LIN {X 0,Y 390.032,Z 462.401,A -85,B 0,C 180,E1 -11489.872,E2 -11489.872} C_VEL
LIN {X 0,Y 390.019,Z 462.384,A -85,B 0,C 180,E1 -11493.227,E2 -11493.227} C_VEL
LIN {X 0,Y 390.057,Z 462.395,A -85,B 0,C 180,E1 -11496.766,E2 -11496.766} C_VEL
LIN {X 0,Y 390.061,Z 462.376,A -85,B 0,C 180,E1 -11499.983,E2 -11499.983} C_VEL
LIN {X 0,Y 390.074,Z 462.387,A -85,B 0,C 180,E1 -11503.247,E2 -11503.247} C_VEL
LIN {X 0,Y 390.188,Z 462.376,A -85,B 0,C 180,E1 -11506.563,E2 -11506.563} C_VEL
LIN {X 0,Y 390.178,Z 462.363,A -85,B 0,C 180,E1 -11510.672,E2 -11510.672} C_VEL
LIN {X 0,Y 390.269,Z 462.37,A -85,B 0,C 180,E1 -11513.799,E2 -11513.799} C_VEL
LIN {X 0,Y 390.398,Z 462.338,A -85,B 0,C 180,E1 -11517.938,E2 -11517.938} C_VEL
LIN {X 0,Y 390.398,Z 462.347,A -85,B 0,C 180,E1 -11522.065,E2 -11522.065} C_VEL
LIN {X 0,Y 390.271,Z 462.365,A -85,B 0,C 180,E1 -11526.204,E2 -11526.204} C_VEL
LIN {X 0,Y 390.181,Z 462.355,A -85,B 0,C 180,E1 -11529.331,E2 -11529.331} C_VEL
LIN {X 0,Y 390.151,Z 462.381,A -85,B 0,C 180,E1 -11532.485,E2 -11532.485} C_VEL
LIN {X 0,Y 390.051,Z 462.394,A -85,B 0,C 180,E1 -11535.682,E2 -11535.682} C_VEL
LIN {X 0,Y 390.037,Z 462.377,A -85,B 0,C 180,E1 -11538.927,E2 -11538.927} C_VEL
LIN {X 0,Y 390.029,Z 462.4,A -85,B 0,C 180,E1 -11542.236,E2 -11542.236} C_VEL
LIN {X 0,Y 390.05,Z 462.383,A -85,B 0,C 180,E1 -11545.723,E2 -11545.723} C_VEL
LIN {X 0,Y 390.023,Z 462.396,A -85,B 0,C 180,E1 -11549.114,E2 -11549.114} C_VEL
LIN {X 0,Y 390.041,Z 462.389,A -85,B 0,C 180,E1 -11552.723,E2 -11552.723} C_VEL
LIN {X 0,Y 390.042,Z 462.395,A -85,B 0,C 180,E1 -11555.823,E2 -11555.823} C_VEL
LIN {X 0,Y 390.034,Z 462.394,A -85,B 0,C 180,E1 -11559.213,E2 -11559.213} C_VEL
LIN {X 0,Y 390.03,Z 462.4,A -85,B 0,C 180,E1 -11562.373,E2 -11562.373} C_VEL
LIN {X 0,Y 390.039,Z 462.397,A -85,B 0,C 180,E1 -11565.354,E2 -11565.354} C_VEL
LIN {X 0,Y 390.013,Z 462.387,A -85,B 0,C 180,E1 -11568.185,E2 -11568.185} C_VEL
LIN {X 0,Y 390.056,Z 462.395,A -85,B 0,C 180,E1 -11570.904,E2 -11570.904} C_VEL
LIN {X 0,Y 390.07,Z 462.391,A -85,B 0,C 180,E1 -11574.792,E2 -11574.792} C_VEL
LIN {X 0,Y 390.024,Z 462.406,A -85,B 0,C 180,E1 -11578.496,E2 -11578.496} C_VEL
LIN {X 0,Y 390.119,Z 462.589,A -85,B 0,C 180,E1 -11579.67,E2 -11579.67} C_VEL
LIN {X 0,Y 392.065,Z 472.624,A -85,B 0,C 180,E1 -11582.8,E2 -11582.8} C_VEL
LIN {X 0,Y 392.806,Z 477.057,A -85,B 0,C 180,E1 -11584.071,E2 -11584.071} C_VEL
LIN {X 0,Y 392.549,Z 483.032,A -85,B 0,C 180,E1 -11585.684,E2 -11585.684} C_VEL
LIN {X 0,Y 391.661,Z 493.141,A -85,B 0,C 180,E1 -11588.417,E2 -11588.417} C_VEL
LIN {X 0,Y 391.382,Z 497.053,A -85,B 0,C 180,E1 -11589.469,E2 -11589.469} C_VEL
LIN {X 0,Y 391.927,Z 500.233,A -85,B 0,C 180,E1 -11589.618,E2 -11589.618} C_VEL
LIN {X 0,Y 396.826,Z 527.349,A -85,B 0,C 180,E1 -11590.388,E2 -11590.388} C_VEL
LIN {X 0,Y 395.882,Z 602.023,A -85,B 0,C 180,E1 -11591.767,E2 -11591.767} C_VEL
LIN {X 0,Y 395.479,Z 611.939,A -85,B 0,C 180,E1 -11592.049,E2 -11592.049} C_VEL
LIN {X 0,Y 395.02,Z 621.929,A -85,B 0,C 180,E1 -11592.462,E2 -11592.462} C_VEL
LIN {X 0,Y 394.399,Z 630.315,A -85,B 0,C 180,E1 -11592.901,E2 -11592.901} C_VEL
LIN {X 0,Y 393.654,Z 641.432,A -85,B 0,C 180,E1 -11593.669,E2 -11593.669} C_VEL
LIN {X 0,Y 392.916,Z 650.435,A -85,B 0,C 180,E1 -11594.437,E2 -11594.437} C_VEL
LIN {X 0,Y 392.266,Z 658.483,A -85,B 0,C 180,E1 -11595.259,E2 -11595.259} C_VEL
LIN {X 0,Y 391.546,Z 666.812,A -85,B 0,C 180,E1 -11596.274,E2 -11596.274} C_VEL
LIN {X 0,Y 390.769,Z 675.386,A -85,B 0,C 180,E1 -11597.536,E2 -11597.536} C_VEL
LIN {X 0,Y 390.167,Z 681.375,A -85,B 0,C 180,E1 -11598.572,E2 -11598.572} C_VEL
LIN {X 0,Y 389.667,Z 687.688,A -85,B 0,C 180,E1 -11599.872,E2 -11599.872} C_VEL
LIN {X 0,Y 389.264,Z 692.963,A -85,B 0,C 180,E1 -11601.172,E2 -11601.172} C_VEL
LIN {X 0,Y 388.944,Z 698.057,A -85,B 0,C 180,E1 -11602.734,E2 -11602.734} C_VEL
LIN {X 0,Y 388.73,Z 701.925,A -85,B 0,C 180,E1 -11604.248,E2 -11604.248} C_VEL
LIN {X 0,Y 388.702,Z 704.954,A -85,B 0,C 180,E1 -11605.853,E2 -11605.853} C_VEL
LIN {X 0,Y 388.636,Z 706.452,A -85,B 0,C 180,E1 -11606.89,E2 -11606.89} C_VEL
LIN {X 0,Y 388.705,Z 707.976,A -85,B 0,C 180,E1 -11608.964,E2 -11608.964} C_VEL
LIN {X 0,Y 388.709,Z 708.254,A -85,B 0,C 180,E1 -11610,E2 -11610} C_VEL
LIN {X 0,Y 388.663,Z 707.38,A -85,B 0,C 180,E1 -11612.073,E2 -11612.073} C_VEL
LIN {X 0,Y 388.636,Z 706.452,A -85,B 0,C 180,E1 -11613.11,E2 -11613.11} C_VEL
LIN {X 0,Y 388.744,Z 703.109,A -85,B 0,C 180,E1 -11615.186,E2 -11615.186} C_VEL
LIN {X 0,Y 388.848,Z 699.484,A -85,B 0,C 180,E1 -11616.747,E2 -11616.747} C_VEL
LIN {X 0,Y 389.146,Z 694.753,A -85,B 0,C 180,E1 -11618.307,E2 -11618.307} C_VEL
LIN {X 0,Y 389.578,Z 688.781,A -85,B 0,C 180,E1 -11619.868,E2 -11619.868} C_VEL
LIN {X 0,Y 390.051,Z 682.688,A -85,B 0,C 180,E1 -11621.168,E2 -11621.168} C_VEL
LIN {X 0,Y 390.631,Z 676.947,A -85,B 0,C 180,E1 -11622.204,E2 -11622.204} C_VEL
LIN {X 0,Y 391.252,Z 670.29,A -85,B 0,C 180,E1 -11623.24,E2 -11623.24} C_VEL
LIN {X 0,Y 391.877,Z 663.503,A -85,B 0,C 180,E1 -11624.15,E2 -11624.15} C_VEL
LIN {X 0,Y 392.529,Z 654.768,A -85,B 0,C 180,E1 -11625.14,E2 -11625.14} C_VEL
LIN {X 0,Y 393.366,Z 644.611,A -85,B 0,C 180,E1 -11626.077,E2 -11626.077} C_VEL
LIN {X 0,Y 394.089,Z 636.223,A -85,B 0,C 180,E1 -11626.712,E2 -11626.712} C_VEL
LIN {X 0,Y 394.727,Z 625.715,A -85,B 0,C 180,E1 -11627.351,E2 -11627.351} C_VEL
LIN {X 0,Y 395.28,Z 615.382,A -85,B 0,C 180,E1 -11627.827,E2 -11627.827} C_VEL
LIN {X 0,Y 395.748,Z 604.664,A -85,B 0,C 180,E1 -11628.173,E2 -11628.173} C_VEL
LIN {X 0,Y 396.177,Z 585.472,A -85,B 0,C 180,E1 -11628.554,E2 -11628.554} C_VEL
LIN {X 0,Y 396.727,Z 526.888,A -85,B 0,C 180,E1 -11629.626,E2 -11629.626} C_VEL
LIN {X 0,Y 391.632,Z 498.91,A -85,B 0,C 180,E1 -11630.424,E2 -11630.424} C_VEL
LIN {X 0,Y 391.346,Z 497.047,A -85,B 0,C 180,E1 -11630.533,E2 -11630.533} C_VEL
LIN {X 0,Y 392.557,Z 483.234,A -85,B 0,C 180,E1 -11634.316,E2 -11634.316} C_VEL
LIN {X 0,Y 392.862,Z 477.28,A -85,B 0,C 180,E1 -11635.937,E2 -11635.937} C_VEL
LIN {X 0,Y 391.203,Z 468.061,A -85,B 0,C 180,E1 -11638.625,E2 -11638.625} C_VEL
LIN {X 0,Y 390.098,Z 462.508,A -85,B 0,C 180,E1 -11640.369,E2 -11640.369} C_VEL
LIN {X 0,Y 390.072,Z 462.397,A -85,B 0,C 180,E1 -11644.024,E2 -11644.024} C_VEL
LIN {X 0,Y 390.036,Z 462.399,A -85,B 0,C 180,E1 -11647.78,E2 -11647.78} C_VEL
LIN {X 0,Y 390.016,Z 462.382,A -85,B 0,C 180,E1 -11650.813,E2 -11650.813} C_VEL
LIN {X 0,Y 390.042,Z 462.401,A -85,B 0,C 180,E1 -11653.883,E2 -11653.883} C_VEL
LIN {X 0,Y 390.048,Z 462.396,A -85,B 0,C 180,E1 -11656.787,E2 -11656.787} C_VEL
LIN {X 0,Y 390.01,Z 462.399,A -85,B 0,C 180,E1 -11659.553,E2 -11659.553} C_VEL
LIN {X 0,Y 390.037,Z 462.401,A -85,B 0,C 180,E1 -11662.45,E2 -11662.45} C_VEL
LIN {X 0,Y 390.062,Z 462.383,A -85,B 0,C 180,E1 -11666.043,E2 -11666.043} C_VEL
LIN {X 0,Y 390.043,Z 462.401,A -85,B 0,C 180,E1 -11669.869,E2 -11669.869} C_VEL
LIN {X 0,Y 390.029,Z 462.38,A -85,B 0,C 180,E1 -11673.224,E2 -11673.224} C_VEL
LIN {X 0,Y 390.058,Z 462.394,A -85,B 0,C 180,E1 -11676.766,E2 -11676.766} C_VEL
LIN {X 0,Y 390.066,Z 462.382,A -85,B 0,C 180,E1 -11679.98,E2 -11679.98} C_VEL
LIN {X 0,Y 390.076,Z 462.38,A -85,B 0,C 180,E1 -11683.244,E2 -11683.244} C_VEL
LIN {X 0,Y 390.13,Z 462.384,A -85,B 0,C 180,E1 -11686.599,E2 -11686.599} C_VEL
LIN {X 0,Y 390.152,Z 462.367,A -85,B 0,C 180,E1 -11689.621,E2 -11689.621} C_VEL
LIN {X 0,Y 390.242,Z 462.365,A -85,B 0,C 180,E1 -11692.756,E2 -11692.756} C_VEL
LIN {X 0,Y 390.193,Z 462.378,A -85,B 0,C 180,E1 -11694.832,E2 -11694.832} C_VEL
LIN {X 0,Y 390.399,Z 462.347,A -85,B 0,C 180,E1 -11697.935,E2 -11697.935} C_VEL
LIN {X 0,Y 390.398,Z 462.338,A -85,B 0,C 180,E1 -11702.062,E2 -11702.062} C_VEL
LIN {X 0,Y 390.247,Z 462.37,A -85,B 0,C 180,E1 -11706.515,E2 -11706.515} C_VEL
LIN {X 0,Y 390.178,Z 462.363,A -85,B 0,C 180,E1 -11709.328,E2 -11709.328} C_VEL
LIN {X 0,Y 390.188,Z 462.376,A -85,B 0,C 180,E1 -11713.437,E2 -11713.437} C_VEL
LIN {X 0,Y 390.063,Z 462.388,A -85,B 0,C 180,E1 -11717.269,E2 -11717.269} C_VEL
LIN {X 0,Y 390.041,Z 462.389,A -85,B 0,C 180,E1 -11721.121,E2 -11721.121} C_VEL
LIN {X 0,Y 390.033,Z 462.397,A -85,B 0,C 180,E1 -11724.482,E2 -11724.482} C_VEL
LIN {X 0,Y 390.005,Z 462.387,A -85,B 0,C 180,E1 -11727.996,E2 -11727.996} C_VEL
LIN {X 0,Y 390.01,Z 462.403,A -85,B 0,C 180,E1 -11731.503,E2 -11731.503} C_VEL
LIN {X 0,Y 390.056,Z 462.384,A -85,B 0,C 180,E1 -11735.207,E2 -11735.207} C_VEL
LIN {X 0,Y 390.044,Z 462.395,A -85,B 0,C 180,E1 -11739.095,E2 -11739.095} C_VEL
LIN {X 0,Y 390.017,Z 462.403,A -85,B 0,C 180,E1 -11742.371,E2 -11742.371} C_VEL
LIN {X 0,Y 390.026,Z 462.395,A -85,B 0,C 180,E1 -11745.352,E2 -11745.352} C_VEL
LIN {X 0,Y 389.997,Z 462.37,A -85,B 0,C 180,E1 -11748.183,E2 -11748.183} C_VEL
LIN {X 0,Y 390.039,Z 462.397,A -85,B 0,C 180,E1 -11750.902,E2 -11750.902} C_VEL
LIN {X 0,Y 390.053,Z 462.376,A -85,B 0,C 180,E1 -11754.79,E2 -11754.79} C_VEL
LIN {X 0,Y 390.006,Z 462.404,A -85,B 0,C 180,E1 -11758.495,E2 -11758.495} C_VEL
LIN {X 0,Y 390,Z 462.399,A -85,B 0,C 180,E1 -11762.002,E2 -11762.002} C_VEL
LIN {X 0,Y 390.027,Z 462.403,A -85,B 0,C 180,E1 -11765.516,E2 -11765.516} C_VEL
LIN {X 0,Y 390.04,Z 462.401,A -85,B 0,C 180,E1 -11768.877,E2 -11768.877} C_VEL
LIN {X 0,Y 390.087,Z 462.397,A -85,B 0,C 180,E1 -11772.165,E2 -11772.165} C_VEL
LIN {X 0,Y 390.076,Z 462.398,A -85,B 0,C 180,E1 -11775.39,E2 -11775.39} C_VEL
LIN {X 0,Y 390.151,Z 462.389,A -85,B 0,C 180,E1 -11777.516,E2 -11777.516} C_VEL
LIN {X 0,Y 390.197,Z 462.441,A -85,B 0,C 180,E1 -11781.324,E2 -11781.324} C_VEL
LIN {X 0,Y 390.388,Z 463.13,A -85,B 0,C 180,E1 -11782.098,E2 -11782.098} C_VEL
LIN {X 0,Y 391.792,Z 466.011,A -85,B 0,C 180,E1 -11783.369,E2 -11783.369} C_VEL
LIN {X 0,Y 393.843,Z 467.786,A -85,B 0,C 180,E1 -11785.138,E2 -11785.138} C_VEL
LIN {X 0,Y 395.352,Z 468.399,A -85,B 0,C 180,E1 -11786.943,E2 -11786.943} C_VEL
LIN {X 0,Y 396.116,Z 469.029,A -85,B 0,C 180,E1 -11788.983,E2 -11788.983} C_VEL
LIN {X 0,Y 396.296,Z 469.069,A -85,B 0,C 180,E1 -11790,E2 -11790} C_VEL
LIN {X 0,Y 395.957,Z 468.754,A -85,B 0,C 180,E1 -11791.78,E2 -11791.78} C_VEL
LIN {X 0,Y 394.887,Z 468.274,A -85,B 0,C 180,E1 -11793.622,E2 -11793.622} C_VEL
LIN {X 0,Y 393.539,Z 467.583,A -85,B 0,C 180,E1 -11795.123,E2 -11795.123} C_VEL
LIN {X 0,Y 391.792,Z 466.011,A -85,B 0,C 180,E1 -11796.631,E2 -11796.631} C_VEL
LIN {X 0,Y 390.503,Z 463.555,A -85,B 0,C 180,E1 -11797.722,E2 -11797.722} C_VEL
LIN {X 0,Y 390.256,Z 462.638,A -85,B 0,C 180,E1 -11798.283,E2 -11798.283} C_VEL
LIN {X 0,Y 390.121,Z 462.392,A -85,B 0,C 180,E1 -11801.429,E2 -11801.429} C_VEL
LIN {X 0,Y 390.153,Z 462.388,A -85,B 0,C 180,E1 -11803.543,E2 -11803.543} C_VEL
LIN {X 0,Y 390.092,Z 462.395,A -85,B 0,C 180,E1 -11807.288,E2 -11807.288} C_VEL
LIN {X 0,Y 390.072,Z 462.398,A -85,B 0,C 180,E1 -11810.47,E2 -11810.47} C_VEL
LIN {X 0,Y 390.047,Z 462.401,A -85,B 0,C 180,E1 -11813.353,E2 -11813.353} C_VEL
LIN {X 0,Y 390.015,Z 462.403,A -85,B 0,C 180,E1 -11816.775,E2 -11816.775} C_VEL
LIN {X 0,Y 390.021,Z 462.393,A -85,B 0,C 180,E1 -11820.301,E2 -11820.301} C_VEL
LIN {X 0,Y 389.994,Z 462.397,A -85,B 0,C 180,E1 -11820.778,E2 -11820.778} C_VEL
LIN {X 0,Y 389.32,Z 462.491,A -85,B 0,C 180,E1 -11821.641,E2 -11821.641} C_VEL
LIN {X 0,Y 386.473,Z 462.838,A -85,B 0,C 180,E1 -11823.042,E2 -11823.042} C_VEL
LIN {X 0,Y 384.074,Z 463.124,A -85,B 0,C 180,E1 -11824.175,E2 -11824.175} C_VEL
LIN {X 0,Y 383.052,Z 463.246,A -85,B 0,C 180,E1 -11825.051,E2 -11825.051} C_VEL
LIN {X 0,Y 382.973,Z 463.257,A -85,B 0,C 180,E1 -11825.348,E2 -11825.348} C_VEL
LIN {X 0,Y 382.963,Z 463.279,A -85,B 0,C 180,E1 -11828.605,E2 -11828.605} C_VEL
LIN {X 0,Y 382.945,Z 463.25,A -85,B 0,C 180,E1 -11831.352,E2 -11831.352} C_VEL
LIN {X 0,Y 382.974,Z 463.266,A -85,B 0,C 180,E1 -11834.303,E2 -11834.303} C_VEL
LIN {X 0,Y 382.969,Z 463.279,A -85,B 0,C 180,E1 -11837.237,E2 -11837.237} C_VEL
LIN {X 0,Y 382.972,Z 463.277,A -85,B 0,C 180,E1 -11840.421,E2 -11840.421} C_VEL
LIN {X 0,Y 383.001,Z 463.268,A -85,B 0,C 180,E1 -11844.044,E2 -11844.044} C_VEL
LIN {X 0,Y 382.974,Z 463.276,A -85,B 0,C 180,E1 -11847.58,E2 -11847.58} C_VEL
LIN {X 0,Y 382.964,Z 463.275,A -85,B 0,C 180,E1 -11850.3,E2 -11850.3} C_VEL
LIN {X 0,Y 382.993,Z 463.267,A -85,B 0,C 180,E1 -11854.047,E2 -11854.047} C_VEL
LIN {X 0,Y 382.979,Z 463.278,A -85,B 0,C 180,E1 -11857.335,E2 -11857.335} C_VEL
LIN {X 0,Y 383.003,Z 463.251,A -85,B 0,C 180,E1 -11860.715,E2 -11860.715} C_VEL
LIN {X 0,Y 383.002,Z 463.276,A -85,B 0,C 180,E1 -11864.025,E2 -11864.025} C_VEL
LIN {X 0,Y 383.127,Z 463.255,A -85,B 0,C 180,E1 -11867.285,E2 -11867.285} C_VEL
LIN {X 0,Y 383.129,Z 463.238,A -85,B 0,C 180,E1 -11870.499,E2 -11870.499} C_VEL
LIN {X 0,Y 383.227,Z 463.246,A -85,B 0,C 180,E1 -11873.684,E2 -11873.684} C_VEL
LIN {X 0,Y 383.363,Z 463.214,A -85,B 0,C 180,E1 -11877.9,E2 -11877.9} C_VEL
LIN {X 0,Y 383.363,Z 463.223,A -85,B 0,C 180,E1 -11882.103,E2 -11882.103} C_VEL
LIN {X 0,Y 383.229,Z 463.241,A -85,B 0,C 180,E1 -11886.319,E2 -11886.319} C_VEL
LIN {X 0,Y 383.171,Z 463.23,A -85,B 0,C 180,E1 -11888.439,E2 -11888.439} C_VEL
LIN {X 0,Y 383.079,Z 463.254,A -85,B 0,C 180,E1 -11891.644,E2 -11891.644} C_VEL
LIN {X 0,Y 383.05,Z 463.27,A -85,B 0,C 180,E1 -11893.8,E2 -11893.8} C_VEL
LIN {X 0,Y 383.02,Z 463.256,A -85,B 0,C 180,E1 -11897.421,E2 -11897.421} C_VEL
LIN {X 0,Y 383.01,Z 463.267,A -85,B 0,C 180,E1 -11900.641,E2 -11900.641} C_VEL
LIN {X 0,Y 383.007,Z 463.274,A -85,B 0,C 180,E1 -11903.81,E2 -11903.81} C_VEL
LIN {X 0,Y 382.968,Z 463.26,A -85,B 0,C 180,E1 -11907.31,E2 -11907.31} C_VEL
LIN {X 0,Y 382.981,Z 463.276,A -85,B 0,C 180,E1 -11910.92,E2 -11910.92} C_VEL
LIN {X 0,Y 383.012,Z 463.265,A -85,B 0,C 180,E1 -11914.67,E2 -11914.67} C_VEL
LIN {X 0,Y 382.991,Z 463.277,A -85,B 0,C 180,E1 -11917.903,E2 -11917.903} C_VEL
LIN {X 0,Y 382.961,Z 463.278,A -85,B 0,C 180,E1 -11921.352,E2 -11921.352} C_VEL
LIN {X 0,Y 382.989,Z 463.273,A -85,B 0,C 180,E1 -11924.303,E2 -11924.303} C_VEL
LIN {X 0,Y 382.982,Z 463.277,A -85,B 0,C 180,E1 -11927.237,E2 -11927.237} C_VEL
LIN {X 0,Y 382.986,Z 463.269,A -85,B 0,C 180,E1 -11930.42,E2 -11930.42} C_VEL
LIN {X 0,Y 383.014,Z 463.264,A -85,B 0,C 180,E1 -11934.044,E2 -11934.044} C_VEL
LIN {X 0,Y 382.985,Z 463.272,A -85,B 0,C 180,E1 -11937.58,E2 -11937.58} C_VEL
LIN {X 0,Y 383.068,Z 463.508,A -85,B 0,C 180,E1 -11939.384,E2 -11939.384} C_VEL
LIN {X 0,Y 385.013,Z 473.48,A -85,B 0,C 180,E1 -11942.554,E2 -11942.554} C_VEL
LIN {X 0,Y 385.9,Z 479.744,A -85,B 0,C 180,E1 -11944.372,E2 -11944.372} C_VEL
LIN {X 0,Y 384.943,Z 490.991,A -85,B 0,C 180,E1 -11947.456,E2 -11947.456} C_VEL
LIN {X 0,Y 384.447,Z 496.846,A -85,B 0,C 180,E1 -11949.081,E2 -11949.081} C_VEL
LIN {X 0,Y 385.014,Z 500.013,A -85,B 0,C 180,E1 -11949.235,E2 -11949.235} C_VEL
LIN {X 0,Y 389.987,Z 527.524,A -85,B 0,C 180,E1 -11950.037,E2 -11950.037} C_VEL
LIN {X 0,Y 389.957,Z 544.905,A -85,B 0,C 180,E1 -11950.368,E2 -11950.368} C_VEL
LIN {X 0,Y 389.156,Z 601.827,A -85,B 0,C 180,E1 -11951.44,E2 -11951.44} C_VEL
LIN {X 0,Y 388.725,Z 611.743,A -85,B 0,C 180,E1 -11951.726,E2 -11951.726} C_VEL
LIN {X 0,Y 388.253,Z 621.733,A -85,B 0,C 180,E1 -11952.146,E2 -11952.146} C_VEL
LIN {X 0,Y 387.504,Z 632.088,A -85,B 0,C 180,E1 -11952.723,E2 -11952.723} C_VEL
LIN {X 0,Y 386.829,Z 641.235,A -85,B 0,C 180,E1 -11953.373,E2 -11953.373} C_VEL
LIN {X 0,Y 386.047,Z 650.238,A -85,B 0,C 180,E1 -11954.153,E2 -11954.153} C_VEL
LIN {X 0,Y 385.326,Z 658.968,A -85,B 0,C 180,E1 -11955.071,E2 -11955.071} C_VEL
LIN {X 0,Y 384.598,Z 666.804,A -85,B 0,C 180,E1 -11956.048,E2 -11956.048} C_VEL
LIN {X 0,Y 383.824,Z 675.189,A -85,B 0,C 180,E1 -11957.307,E2 -11957.307} C_VEL
LIN {X 0,Y 383.183,Z 681.178,A -85,B 0,C 180,E1 -11958.361,E2 -11958.361} C_VEL
LIN {X 0,Y 382.663,Z 687.492,A -85,B 0,C 180,E1 -11959.685,E2 -11959.685} C_VEL
LIN {X 0,Y 382.219,Z 692.766,A -85,B 0,C 180,E1 -11961.008,E2 -11961.008} C_VEL
LIN {X 0,Y 381.873,Z 697.86,A -85,B 0,C 180,E1 -11962.598,E2 -11962.598} C_VEL
LIN {X 0,Y 381.674,Z 701.247,A -85,B 0,C 180,E1 -11963.907,E2 -11963.907} C_VEL
LIN {X 0,Y 381.627,Z 704.758,A -85,B 0,C 180,E1 -11965.776,E2 -11965.776} C_VEL
LIN {X 0,Y 381.548,Z 706.256,A -85,B 0,C 180,E1 -11966.832,E2 -11966.832} C_VEL
LIN {X 0,Y 381.604,Z 707.779,A -85,B 0,C 180,E1 -11968.945,E2 -11968.945} C_VEL
LIN {X 0,Y 381.623,Z 708.059,A -85,B 0,C 180,E1 -11970,E2 -11970} C_VEL
LIN {X 0,Y 381.561,Z 707.183,A -85,B 0,C 180,E1 -11972.111,E2 -11972.111} C_VEL
LIN {X 0,Y 381.548,Z 706.256,A -85,B 0,C 180,E1 -11973.168,E2 -11973.168} C_VEL
LIN {X 0,Y 381.644,Z 702.912,A -85,B 0,C 180,E1 -11975.283,E2 -11975.283} C_VEL
LIN {X 0,Y 381.785,Z 699.287,A -85,B 0,C 180,E1 -11976.872,E2 -11976.872} C_VEL
LIN {X 0,Y 382.099,Z 694.556,A -85,B 0,C 180,E1 -11978.461,E2 -11978.461} C_VEL
LIN {X 0,Y 382.541,Z 688.584,A -85,B 0,C 180,E1 -11980.051,E2 -11980.051} C_VEL
LIN {X 0,Y 383.064,Z 682.491,A -85,B 0,C 180,E1 -11981.375,E2 -11981.375} C_VEL
LIN {X 0,Y 383.647,Z 676.75,A -85,B 0,C 180,E1 -11982.43,E2 -11982.43} C_VEL
LIN {X 0,Y 384.311,Z 670.093,A -85,B 0,C 180,E1 -11983.483,E2 -11983.483} C_VEL
LIN {X 0,Y 385.024,Z 662.625,A -85,B 0,C 180,E1 -11984.491,E2 -11984.491} C_VEL
LIN {X 0,Y 385.705,Z 654.177,A -85,B 0,C 180,E1 -11985.455,E2 -11985.455} C_VEL
LIN {X 0,Y 386.557,Z 644.415,A -85,B 0,C 180,E1 -11986.368,E2 -11986.368} C_VEL
LIN {X 0,Y 387.29,Z 636.027,A -85,B 0,C 180,E1 -11987.014,E2 -11987.014} C_VEL
LIN {X 0,Y 387.967,Z 625.519,A -85,B 0,C 180,E1 -11987.663,E2 -11987.663} C_VEL
LIN {X 0,Y 388.529,Z 615.186,A -85,B 0,C 180,E1 -11988.147,E2 -11988.147} C_VEL
LIN {X 0,Y 389.02,Z 604.468,A -85,B 0,C 180,E1 -11988.498,E2 -11988.498} C_VEL
LIN {X 0,Y 389.471,Z 583.485,A -85,B 0,C 180,E1 -11988.92,E2 -11988.92} C_VEL
LIN {X 0,Y 390.114,Z 528.302,A -85,B 0,C 180,E1 -11989.942,E2 -11989.942} C_VEL
LIN {X 0,Y 384.978,Z 500.003,A -85,B 0,C 180,E1 -11990.768,E2 -11990.768} C_VEL
LIN {X 0,Y 384.4,Z 497.123,A -85,B 0,C 180,E1 -11990.887,E2 -11990.887} C_VEL
LIN {X 0,Y 384.468,Z 495.674,A -85,B 0,C 180,E1 -11991.206,E2 -11991.206} C_VEL
LIN {X 0,Y 385.712,Z 483.045,A -85,B 0,C 180,E1 -11994.776,E2 -11994.776} C_VEL
LIN {X 0,Y 385.919,Z 478.968,A -85,B 0,C 180,E1 -11995.917,E2 -11995.917} C_VEL
LIN {X 0,Y 384.343,Z 469.806,A -85,B 0,C 180,E1 -11998.63,E2 -11998.63} C_VEL
LIN {X 0,Y 383.04,Z 463.38,A -85,B 0,C 180,E1 -12000.692,E2 -12000.692} C_VEL
LIN {X 0,Y 383.019,Z 463.277,A -85,B 0,C 180,E1 -12004.338,E2 -12004.338} C_VEL
LIN {X 0,Y 382.991,Z 463.274,A -85,B 0,C 180,E1 -12007.269,E2 -12007.269} C_VEL
LIN {X 0,Y 382.975,Z 463.264,A -85,B 0,C 180,E1 -12009.962,E2 -12009.962} C_VEL
LIN {X 0,Y 383.009,Z 463.273,A -85,B 0,C 180,E1 -12012.778,E2 -12012.778} C_VEL
LIN {X 0,Y 382.99,Z 463.273,A -85,B 0,C 180,E1 -12015.787,E2 -12015.787} C_VEL
LIN {X 0,Y 382.962,Z 463.277,A -85,B 0,C 180,E1 -12018.8,E2 -12018.8} C_VEL
LIN {X 0,Y 382.991,Z 463.277,A -85,B 0,C 180,E1 -12022.097,E2 -12022.097} C_VEL
LIN {X 0,Y 383.012,Z 463.265,A -85,B 0,C 180,E1 -12025.33,E2 -12025.33} C_VEL
LIN {X 0,Y 382.981,Z 463.276,A -85,B 0,C 180,E1 -12029.08,E2 -12029.08} C_VEL
LIN {X 0,Y 382.968,Z 463.26,A -85,B 0,C 180,E1 -12032.69,E2 -12032.69} C_VEL
LIN {X 0,Y 383.007,Z 463.274,A -85,B 0,C 180,E1 -12036.19,E2 -12036.19} C_VEL
LIN {X 0,Y 383.033,Z 463.265,A -85,B 0,C 180,E1 -12039.596,E2 -12039.596} C_VEL
LIN {X 0,Y 383.035,Z 463.257,A -85,B 0,C 180,E1 -12042.927,E2 -12042.927} C_VEL
LIN {X 0,Y 383.088,Z 463.262,A -85,B 0,C 180,E1 -12046.485,E2 -12046.485} C_VEL
LIN {X 0,Y 383.116,Z 463.245,A -85,B 0,C 180,E1 -12049.428,E2 -12049.428} C_VEL
LIN {X 0,Y 383.197,Z 463.242,A -85,B 0,C 180,E1 -12052.622,E2 -12052.622} C_VEL
LIN {X 0,Y 383.165,Z 463.254,A -85,B 0,C 180,E1 -12054.736,E2 -12054.736} C_VEL
LIN {X 0,Y 383.364,Z 463.223,A -85,B 0,C 180,E1 -12057.897,E2 -12057.897} C_VEL
LIN {X 0,Y 383.363,Z 463.214,A -85,B 0,C 180,E1 -12062.1,E2 -12062.1} C_VEL
LIN {X 0,Y 383.211,Z 463.246,A -85,B 0,C 180,E1 -12066.504,E2 -12066.504} C_VEL
LIN {X 0,Y 383.129,Z 463.238,A -85,B 0,C 180,E1 -12069.501,E2 -12069.501} C_VEL
LIN {X 0,Y 383.119,Z 463.257,A -85,B 0,C 180,E1 -12073.534,E2 -12073.534} C_VEL
LIN {X 0,Y 383.016,Z 463.267,A -85,B 0,C 180,E1 -12077.419,E2 -12077.419} C_VEL
LIN {X 0,Y 383.005,Z 463.264,A -85,B 0,C 180,E1 -12080.639,E2 -12080.639} C_VEL
LIN {X 0,Y 383.001,Z 463.278,A -85,B 0,C 180,E1 -12083.807,E2 -12083.807} C_VEL
LIN {X 0,Y 382.958,Z 463.262,A -85,B 0,C 180,E1 -12087.307,E2 -12087.307} C_VEL
LIN {X 0,Y 382.97,Z 463.279,A -85,B 0,C 180,E1 -12090.917,E2 -12090.917} C_VEL
LIN {X 0,Y 382.999,Z 463.262,A -85,B 0,C 180,E1 -12094.667,E2 -12094.667} C_VEL
LIN {X 0,Y 382.979,Z 463.282,A -85,B 0,C 180,E1 -12097.901,E2 -12097.901} C_VEL
LIN {X 0,Y 382.947,Z 463.271,A -85,B 0,C 180,E1 -12101.349,E2 -12101.349} C_VEL
LIN {X 0,Y 382.975,Z 463.277,A -85,B 0,C 180,E1 -12104.301,E2 -12104.301} C_VEL
LIN {X 0,Y 382.967,Z 463.248,A -85,B 0,C 180,E1 -12107.235,E2 -12107.235} C_VEL
LIN {X 0,Y 382.969,Z 463.271,A -85,B 0,C 180,E1 -12110.418,E2 -12110.418} C_VEL
LIN {X 0,Y 382.998,Z 463.261,A -85,B 0,C 180,E1 -12114.042,E2 -12114.042} C_VEL
LIN {X 0,Y 382.97,Z 463.278,A -85,B 0,C 180,E1 -12117.578,E2 -12117.578} C_VEL
LIN {X 0,Y 382.959,Z 463.266,A -85,B 0,C 180,E1 -12120.298,E2 -12120.298} C_VEL
LIN {X 0,Y 382.987,Z 463.281,A -85,B 0,C 180,E1 -12124.044,E2 -12124.044} C_VEL
LIN {X 0,Y 382.974,Z 463.282,A -85,B 0,C 180,E1 -12127.333,E2 -12127.333} C_VEL
LIN {X 0,Y 383.04,Z 463.274,A -85,B 0,C 180,E1 -12130.715,E2 -12130.715} C_VEL
LIN {X 0,Y 383.004,Z 463.279,A -85,B 0,C 180,E1 -12134.024,E2 -12134.024} C_VEL
LIN {X 0,Y 383.118,Z 463.264,A -85,B 0,C 180,E1 -12137.283,E2 -12137.283} C_VEL
LIN {X 0,Y 383.139,Z 463.583,A -85,B 0,C 180,E1 -12138.56,E2 -12138.56} C_VEL
LIN {X 0,Y 383.428,Z 464.757,A -85,B 0,C 180,E1 -12138.971,E2 -12138.971} C_VEL
LIN {X 0,Y 384.572,Z 466.794,A -85,B 0,C 180,E1 -12139.603,E2 -12139.603} C_VEL
LIN {X 0,Y 386.855,Z 468.647,A -85,B 0,C 180,E1 -12140.722,E2 -12140.722} C_VEL
LIN {X 0,Y 388.802,Z 469.821,A -85,B 0,C 180,E1 -12141.834,E2 -12141.834} C_VEL
LIN {X 0,Y 390.416,Z 472.61,A -85,B 0,C 180,E1 -12143.021,E2 -12143.021} C_VEL
LIN {X 0,Y 391.927,Z 474.117,A -85,B 0,C 180,E1 -12144.211,E2 -12144.211} C_VEL
LIN {X 0,Y 393.427,Z 475.106,A -85,B 0,C 180,E1 -12145.646,E2 -12145.646} C_VEL
LIN {X 0,Y 394.712,Z 475.569,A -85,B 0,C 180,E1 -12147.449,E2 -12147.449} C_VEL
LIN {X 0,Y 395.254,Z 476.076,A -85,B 0,C 180,E1 -12148.981,E2 -12148.981} C_VEL
LIN {X 0,Y 395.432,Z 476.106,A -85,B 0,C 180,E1 -12150,E2 -12150} C_VEL
LIN {X 0,Y 395.09,Z 475.808,A -85,B 0,C 180,E1 -12151.784,E2 -12151.784} C_VEL
LIN {X 0,Y 394.236,Z 475.37,A -85,B 0,C 180,E1 -12153.375,E2 -12153.375} C_VEL
LIN {X 0,Y 392.647,Z 474.648,A -85,B 0,C 180,E1 -12155.135,E2 -12155.135} C_VEL
LIN {X 0,Y 390.776,Z 473.066,A -85,B 0,C 180,E1 -12156.713,E2 -12156.713} C_VEL
LIN {X 0,Y 389.074,Z 470.321,A -85,B 0,C 180,E1 -12157.995,E2 -12157.995} C_VEL
LIN {X 0,Y 388.296,Z 469.392,A -85,B 0,C 180,E1 -12158.456,E2 -12158.456} C_VEL
LIN {X 0,Y 385.834,Z 468.03,A -85,B 0,C 180,E1 -12159.766,E2 -12159.766} C_VEL
LIN {X 0,Y 383.861,Z 465.743,A -85,B 0,C 180,E1 -12160.783,E2 -12160.783} C_VEL
LIN {X 0,Y 383.168,Z 463.833,A -85,B 0,C 180,E1 -12161.305,E2 -12161.305} C_VEL
LIN {X 0,Y 383.096,Z 463.3,A -85,B 0,C 180,E1 -12161.91,E2 -12161.91} C_VEL
LIN {X 0,Y 383.012,Z 463.278,A -85,B 0,C 180,E1 -12164.885,E2 -12164.885} C_VEL
LIN {X 0,Y 383.031,Z 463.275,A -85,B 0,C 180,E1 -12168.175,E2 -12168.175} C_VEL
LIN {X 0,Y 382.976,Z 463.282,A -85,B 0,C 180,E1 -12171.532,E2 -12171.532} C_VEL
LIN {X 0,Y 382.971,Z 463.281,A -85,B 0,C 180,E1 -12174.966,E2 -12174.966} C_VEL
LIN {X 0,Y 382.96,Z 463.269,A -85,B 0,C 180,E1 -12178.499,E2 -12178.499} C_VEL
LIN {X 0,Y 382.993,Z 463.277,A -85,B 0,C 180,E1 -12182.151,E2 -12182.151} C_VEL
LIN {X 0,Y 382.973,Z 463.257,A -85,B 0,C 180,E1 -12185.348,E2 -12185.348} C_VEL
LIN {X 0,Y 382.324,Z 463.351,A -85,B 0,C 180,E1 -12186.226,E2 -12186.226} C_VEL
LIN {X 0,Y 379.502,Z 463.713,A -85,B 0,C 180,E1 -12187.653,E2 -12187.653} C_VEL
LIN {X 0,Y 377.085,Z 464.012,A -85,B 0,C 180,E1 -12188.807,E2 -12188.807} C_VEL
LIN {X 0,Y 376.021,Z 464.135,A -85,B 0,C 180,E1 -12189.699,E2 -12189.699} C_VEL
LIN {X 0,Y 375.92,Z 464.141,A -85,B 0,C 180,E1 -12190.001,E2 -12190.001} C_VEL
LIN {X 0,Y 375.911,Z 464.136,A -85,B 0,C 180,E1 -12193.768,E2 -12193.768} C_VEL
LIN {X 0,Y 375.919,Z 464.157,A -85,B 0,C 180,E1 -12196.812,E2 -12196.812} C_VEL
LIN {X 0,Y 375.921,Z 464.156,A -85,B 0,C 180,E1 -12200.535,E2 -12200.535} C_VEL
LIN {X 0,Y 375.945,Z 464.155,A -85,B 0,C 180,E1 -12203.499,E2 -12203.499} C_VEL
LIN {X 0,Y 375.946,Z 464.142,A -85,B 0,C 180,E1 -12205.89,E2 -12205.89} C_VEL
LIN {X 0,Y 375.95,Z 464.157,A -85,B 0,C 180,E1 -12209.688,E2 -12209.688} C_VEL
LIN {X 0,Y 375.907,Z 464.141,A -85,B 0,C 180,E1 -12212.136,E2 -12212.136} C_VEL
LIN {X 0,Y 375.95,Z 464.154,A -85,B 0,C 180,E1 -12215.718,E2 -12215.718} C_VEL
LIN {X 0,Y 375.948,Z 464.144,A -85,B 0,C 180,E1 -12219.197,E2 -12219.197} C_VEL
LIN {X 0,Y 375.971,Z 464.144,A -85,B 0,C 180,E1 -12222.599,E2 -12222.599} C_VEL
LIN {X 0,Y 376.083,Z 464.134,A -85,B 0,C 180,E1 -12226.344,E2 -12226.344} C_VEL
LIN {X 0,Y 376.1,Z 464.111,A -85,B 0,C 180,E1 -12230.32,E2 -12230.32} C_VEL
LIN {X 0,Y 376.187,Z 464.122,A -85,B 0,C 180,E1 -12233.566,E2 -12233.566} C_VEL
LIN {X 0,Y 376.327,Z 464.09,A -85,B 0,C 180,E1 -12237.861,E2 -12237.861} C_VEL
LIN {X 0,Y 376.327,Z 464.1,A -85,B 0,C 180,E1 -12242.142,E2 -12242.142} C_VEL
LIN {X 0,Y 376.189,Z 464.116,A -85,B 0,C 180,E1 -12246.438,E2 -12246.438} C_VEL
LIN {X 0,Y 376.103,Z 464.107,A -85,B 0,C 180,E1 -12249.683,E2 -12249.683} C_VEL
LIN {X 0,Y 376.038,Z 464.141,A -85,B 0,C 180,E1 -12253.628,E2 -12253.628} C_VEL
LIN {X 0,Y 375.979,Z 464.13,A -85,B 0,C 180,E1 -12257.578,E2 -12257.578} C_VEL
LIN {X 0,Y 375.978,Z 464.143,A -85,B 0,C 180,E1 -12260.834,E2 -12260.834} C_VEL
LIN {X 0,Y 375.934,Z 464.149,A -85,B 0,C 180,E1 -12264.287,E2 -12264.287} C_VEL
LIN {X 0,Y 375.911,Z 464.137,A -85,B 0,C 180,E1 -12266.662,E2 -12266.662} C_VEL
LIN {X 0,Y 375.913,Z 464.154,A -85,B 0,C 180,E1 -12269.085,E2 -12269.085} C_VEL
LIN {X 0,Y 375.956,Z 464.155,A -85,B 0,C 180,E1 -12271.564,E2 -12271.564} C_VEL
LIN {X 0,Y 375.949,Z 464.146,A -85,B 0,C 180,E1 -12275.418,E2 -12275.418} C_VEL
LIN {X 0,Y 375.933,Z 464.152,A -85,B 0,C 180,E1 -12278.263,E2 -12278.263} C_VEL
LIN {X 0,Y 375.914,Z 464.158,A -85,B 0,C 180,E1 -12281.598,E2 -12281.598} C_VEL
LIN {X 0,Y 375.92,Z 464.155,A -85,B 0,C 180,E1 -12284.731,E2 -12284.731} C_VEL
LIN {X 0,Y 375.908,Z 464.15,A -85,B 0,C 180,E1 -12287.697,E2 -12287.697} C_VEL
LIN {X 0,Y 375.934,Z 464.149,A -85,B 0,C 180,E1 -12290.534,E2 -12290.534} C_VEL
LIN {X 0,Y 375.959,Z 464.143,A -85,B 0,C 180,E1 -12293.498,E2 -12293.498} C_VEL
LIN {X 0,Y 375.96,Z 464.155,A -85,B 0,C 180,E1 -12295.889,E2 -12295.889} C_VEL
LIN {X 0,Y 376.008,Z 464.333,A -85,B 0,C 180,E1 -12299.042,E2 -12299.042} C_VEL
LIN {X 0,Y 377.99,Z 474.336,A -85,B 0,C 180,E1 -12302.301,E2 -12302.301} C_VEL
LIN {X 0,Y 378.956,Z 480.604,A -85,B 0,C 180,E1 -12304.163,E2 -12304.163} C_VEL
LIN {X 0,Y 378.053,Z 490.795,A -85,B 0,C 180,E1 -12307.022,E2 -12307.022} C_VEL
LIN {X 0,Y 377.522,Z 496.692,A -85,B 0,C 180,E1 -12308.686,E2 -12308.686} C_VEL
LIN {X 0,Y 378.373,Z 501.077,A -85,B 0,C 180,E1 -12308.878,E2 -12308.878} C_VEL
LIN {X 0,Y 383.447,Z 529.25,A -85,B 0,C 180,E1 -12309.719,E2 -12309.719} C_VEL
LIN {X 0,Y 382.438,Z 601.631,A -85,B 0,C 180,E1 -12311.102,E2 -12311.102} C_VEL
LIN {X 0,Y 382.002,Z 611.547,A -85,B 0,C 180,E1 -12311.392,E2 -12311.392} C_VEL
LIN {X 0,Y 381.499,Z 621.536,A -85,B 0,C 180,E1 -12311.819,E2 -12311.819} C_VEL
LIN {X 0,Y 380.714,Z 631.891,A -85,B 0,C 180,E1 -12312.405,E2 -12312.405} C_VEL
LIN {X 0,Y 380.022,Z 641.039,A -85,B 0,C 180,E1 -12313.066,E2 -12313.066} C_VEL
LIN {X 0,Y 379.207,Z 650.041,A -85,B 0,C 180,E1 -12313.859,E2 -12313.859} C_VEL
LIN {X 0,Y 378.434,Z 658.771,A -85,B 0,C 180,E1 -12314.792,E2 -12314.792} C_VEL
LIN {X 0,Y 377.671,Z 666.788,A -85,B 0,C 180,E1 -12315.814,E2 -12315.814} C_VEL
LIN {X 0,Y 376.872,Z 674.992,A -85,B 0,C 180,E1 -12317.069,E2 -12317.069} C_VEL
LIN {X 0,Y 376.214,Z 680.982,A -85,B 0,C 180,E1 -12318.142,E2 -12318.142} C_VEL
LIN {X 0,Y 375.652,Z 687.295,A -85,B 0,C 180,E1 -12319.49,E2 -12319.49} C_VEL
LIN {X 0,Y 375.192,Z 692.569,A -85,B 0,C 180,E1 -12320.838,E2 -12320.838} C_VEL
LIN {X 0,Y 374.809,Z 697.663,A -85,B 0,C 180,E1 -12322.458,E2 -12322.458} C_VEL
LIN {X 0,Y 374.57,Z 701.388,A -85,B 0,C 180,E1 -12323.959,E2 -12323.959} C_VEL
LIN {X 0,Y 374.531,Z 704.562,A -85,B 0,C 180,E1 -12325.695,E2 -12325.695} C_VEL
LIN {X 0,Y 374.463,Z 706.06,A -85,B 0,C 180,E1 -12326.772,E2 -12326.772} C_VEL
LIN {X 0,Y 374.505,Z 707.583,A -85,B 0,C 180,E1 -12328.925,E2 -12328.925} C_VEL
LIN {X 0,Y 374.539,Z 707.863,A -85,B 0,C 180,E1 -12330,E2 -12330} C_VEL
LIN {X 0,Y 374.461,Z 706.987,A -85,B 0,C 180,E1 -12332.151,E2 -12332.151} C_VEL
LIN {X 0,Y 374.463,Z 706.06,A -85,B 0,C 180,E1 -12333.228,E2 -12333.228} C_VEL
LIN {X 0,Y 374.553,Z 702.716,A -85,B 0,C 180,E1 -12335.383,E2 -12335.383} C_VEL
LIN {X 0,Y 374.728,Z 699.091,A -85,B 0,C 180,E1 -12337.002,E2 -12337.002} C_VEL
LIN {X 0,Y 375.041,Z 694.359,A -85,B 0,C 180,E1 -12338.622,E2 -12338.622} C_VEL
LIN {X 0,Y 375.528,Z 688.387,A -85,B 0,C 180,E1 -12340.241,E2 -12340.241} C_VEL
LIN {X 0,Y 376.056,Z 682.293,A -85,B 0,C 180,E1 -12341.59,E2 -12341.59} C_VEL
LIN {X 0,Y 376.69,Z 676.553,A -85,B 0,C 180,E1 -12342.663,E2 -12342.663} C_VEL
LIN {X 0,Y 377.359,Z 669.895,A -85,B 0,C 180,E1 -12343.736,E2 -12343.736} C_VEL
LIN {X 0,Y 378.117,Z 662.427,A -85,B 0,C 180,E1 -12344.762,E2 -12344.762} C_VEL
LIN {X 0,Y 378.854,Z 653.981,A -85,B 0,C 180,E1 -12345.742,E2 -12345.742} C_VEL
LIN {X 0,Y 379.754,Z 644.219,A -85,B 0,C 180,E1 -12346.67,E2 -12346.67} C_VEL
LIN {X 0,Y 380.494,Z 635.83,A -85,B 0,C 180,E1 -12347.328,E2 -12347.328} C_VEL
LIN {X 0,Y 381.215,Z 625.323,A -85,B 0,C 180,E1 -12347.987,E2 -12347.987} C_VEL
LIN {X 0,Y 381.774,Z 614.989,A -85,B 0,C 180,E1 -12348.48,E2 -12348.48} C_VEL
LIN {X 0,Y 382.306,Z 604.273,A -85,B 0,C 180,E1 -12348.835,E2 -12348.835} C_VEL
LIN {X 0,Y 382.769,Z 583.289,A -85,B 0,C 180,E1 -12349.264,E2 -12349.264} C_VEL
LIN {X 0,Y 383.436,Z 529.148,A -85,B 0,C 180,E1 -12350.284,E2 -12350.284} C_VEL
LIN {X 0,Y 378.459,Z 501.649,A -85,B 0,C 180,E1 -12351.106,E2 -12351.106} C_VEL
LIN {X 0,Y 377.489,Z 496.832,A -85,B 0,C 180,E1 -12351.297,E2 -12351.297} C_VEL
LIN {X 0,Y 377.852,Z 492.751,A -85,B 0,C 180,E1 -12352.414,E2 -12352.414} C_VEL
LIN {X 0,Y 378.962,Z 481.853,A -85,B 0,C 180,E1 -12355.542,E2 -12355.542} C_VEL
LIN {X 0,Y 378.321,Z 476.097,A -85,B 0,C 180,E1 -12357.25,E2 -12357.25} C_VEL
LIN {X 0,Y 376.432,Z 466.369,A -85,B 0,C 180,E1 -12360.271,E2 -12360.271} C_VEL
LIN {X 0,Y 375.979,Z 464.226,A -85,B 0,C 180,E1 -12361.082,E2 -12361.082} C_VEL
LIN {X 0,Y 375.978,Z 464.152,A -85,B 0,C 180,E1 -12364.665,E2 -12364.665} C_VEL
LIN {X 0,Y 375.935,Z 464.159,A -85,B 0,C 180,E1 -12368.261,E2 -12368.261} C_VEL
LIN {X 0,Y 375.914,Z 464.14,A -85,B 0,C 180,E1 -12371.596,E2 -12371.596} C_VEL
LIN {X 0,Y 375.919,Z 464.155,A -85,B 0,C 180,E1 -12374.729,E2 -12374.729} C_VEL
LIN {X 0,Y 375.908,Z 464.16,A -85,B 0,C 180,E1 -12377.695,E2 -12377.695} C_VEL
LIN {X 0,Y 375.933,Z 464.149,A -85,B 0,C 180,E1 -12380.532,E2 -12380.532} C_VEL
LIN {X 0,Y 375.957,Z 464.153,A -85,B 0,C 180,E1 -12383.496,E2 -12383.496} C_VEL
LIN {X 0,Y 375.958,Z 464.139,A -85,B 0,C 180,E1 -12385.887,E2 -12385.887} C_VEL
LIN {X 0,Y 375.961,Z 464.153,A -85,B 0,C 180,E1 -12389.686,E2 -12389.686} C_VEL
LIN {X 0,Y 375.917,Z 464.144,A -85,B 0,C 180,E1 -12392.134,E2 -12392.134} C_VEL
LIN {X 0,Y 375.935,Z 464.143,A -85,B 0,C 180,E1 -12394.532,E2 -12394.532} C_VEL
LIN {X 0,Y 375.969,Z 464.149,A -85,B 0,C 180,E1 -12396.885,E2 -12396.885} C_VEL
LIN {X 0,Y 375.955,Z 464.134,A -85,B 0,C 180,E1 -12400.336,E2 -12400.336} C_VEL
LIN {X 0,Y 375.951,Z 464.141,A -85,B 0,C 180,E1 -12403.714,E2 -12403.714} C_VEL
LIN {X 0,Y 376.073,Z 464.134,A -85,B 0,C 180,E1 -12407.039,E2 -12407.039} C_VEL
LIN {X 0,Y 376.103,Z 464.107,A -85,B 0,C 180,E1 -12410.317,E2 -12410.317} C_VEL
LIN {X 0,Y 376.189,Z 464.116,A -85,B 0,C 180,E1 -12413.562,E2 -12413.562} C_VEL
LIN {X 0,Y 376.327,Z 464.1,A -85,B 0,C 180,E1 -12417.858,E2 -12417.858} C_VEL
LIN {X 0,Y 376.327,Z 464.09,A -85,B 0,C 180,E1 -12422.139,E2 -12422.139} C_VEL
LIN {X 0,Y 376.182,Z 464.122,A -85,B 0,C 180,E1 -12426.489,E2 -12426.489} C_VEL
LIN {X 0,Y 376.1,Z 464.111,A -85,B 0,C 180,E1 -12429.68,E2 -12429.68} C_VEL
LIN {X 0,Y 376.083,Z 464.134,A -85,B 0,C 180,E1 -12433.656,E2 -12433.656} C_VEL
LIN {X 0,Y 375.974,Z 464.141,A -85,B 0,C 180,E1 -12437.575,E2 -12437.575} C_VEL
LIN {X 0,Y 375.971,Z 464.141,A -85,B 0,C 180,E1 -12440.83,E2 -12440.83} C_VEL
LIN {X 0,Y 375.95,Z 464.154,A -85,B 0,C 180,E1 -12444.282,E2 -12444.282} C_VEL
LIN {X 0,Y 375.907,Z 464.141,A -85,B 0,C 180,E1 -12447.864,E2 -12447.864} C_VEL
LIN {X 0,Y 375.945,Z 464.156,A -85,B 0,C 180,E1 -12451.561,E2 -12451.561} C_VEL
LIN {X 0,Y 375.937,Z 464.143,A -85,B 0,C 180,E1 -12455.415,E2 -12455.415} C_VEL
LIN {X 0,Y 375.922,Z 464.159,A -85,B 0,C 180,E1 -12458.261,E2 -12458.261} C_VEL
LIN {X 0,Y 375.9,Z 464.15,A -85,B 0,C 180,E1 -12461.596,E2 -12461.596} C_VEL
LIN {X 0,Y 375.906,Z 464.154,A -85,B 0,C 180,E1 -12464.729,E2 -12464.729} C_VEL
LIN {X 0,Y 375.892,Z 464.124,A -85,B 0,C 180,E1 -12467.695,E2 -12467.695} C_VEL
LIN {X 0,Y 375.918,Z 464.151,A -85,B 0,C 180,E1 -12470.532,E2 -12470.532} C_VEL
LIN {X 0,Y 375.942,Z 464.15,A -85,B 0,C 180,E1 -12473.496,E2 -12473.496} C_VEL
LIN {X 0,Y 375.943,Z 464.132,A -85,B 0,C 180,E1 -12475.887,E2 -12475.887} C_VEL
LIN {X 0,Y 375.946,Z 464.145,A -85,B 0,C 180,E1 -12479.686,E2 -12479.686} C_VEL
LIN {X 0,Y 375.902,Z 464.156,A -85,B 0,C 180,E1 -12482.134,E2 -12482.134} C_VEL
LIN {X 0,Y 375.944,Z 464.158,A -85,B 0,C 180,E1 -12485.715,E2 -12485.715} C_VEL
LIN {X 0,Y 375.965,Z 464.155,A -85,B 0,C 180,E1 -12489.196,E2 -12489.196} C_VEL
LIN {X 0,Y 375.998,Z 464.151,A -85,B 0,C 180,E1 -12492.599,E2 -12492.599} C_VEL
LIN {X 0,Y 376.094,Z 464.401,A -85,B 0,C 180,E1 -12496.075,E2 -12496.075} C_VEL
LIN {X 0,Y 376.402,Z 465.541,A -85,B 0,C 180,E1 -12496.467,E2 -12496.467} C_VEL
LIN {X 0,Y 377.859,Z 468.042,A -85,B 0,C 180,E1 -12497.103,E2 -12497.103} C_VEL
LIN {X 0,Y 380.04,Z 469.694,A -85,B 0,C 180,E1 -12497.945,E2 -12497.945} C_VEL
LIN {X 0,Y 381.274,Z 470.628,A -85,B 0,C 180,E1 -12498.47,E2 -12498.47} C_VEL
LIN {X 0,Y 382.756,Z 473.059,A -85,B 0,C 180,E1 -12499.152,E2 -12499.152} C_VEL
LIN {X 0,Y 385.019,Z 475.24,A -85,B 0,C 180,E1 -12500.284,E2 -12500.284} C_VEL
LIN {X 0,Y 387.518,Z 476.739,A -85,B 0,C 180,E1 -12501.625,E2 -12501.625} C_VEL
LIN {X 0,Y 389.138,Z 479.345,A -85,B 0,C 180,E1 -12502.737,E2 -12502.737} C_VEL
LIN {X 0,Y 390.898,Z 481.072,A -85,B 0,C 180,E1 -12504.066,E2 -12504.066} C_VEL
LIN {X 0,Y 392.34,Z 482.031,A -85,B 0,C 180,E1 -12505.377,E2 -12505.377} C_VEL
LIN {X 0,Y 393.608,Z 482.493,A -85,B 0,C 180,E1 -12506.929,E2 -12506.929} C_VEL
LIN {X 0,Y 394.392,Z 483.122,A -85,B 0,C 180,E1 -12508.979,E2 -12508.979} C_VEL
LIN {X 0,Y 394.569,Z 483.133,A -85,B 0,C 180,E1 -12510,E2 -12510} C_VEL
LIN {X 0,Y 394.223,Z 482.858,A -85,B 0,C 180,E1 -12511.788,E2 -12511.788} C_VEL
LIN {X 0,Y 393.608,Z 482.481,A -85,B 0,C 180,E1 -12513.071,E2 -12513.071} C_VEL
LIN {X 0,Y 392.06,Z 481.895,A -85,B 0,C 180,E1 -12514.884,E2 -12514.884} C_VEL
LIN {X 0,Y 389.855,Z 480.205,A -85,B 0,C 180,E1 -12516.729,E2 -12516.729} C_VEL
LIN {X 0,Y 388.054,Z 477.696,A -85,B 0,C 180,E1 -12518.036,E2 -12518.036} C_VEL
LIN {X 0,Y 387.117,Z 476.318,A -85,B 0,C 180,E1 -12518.614,E2 -12518.614} C_VEL
LIN {X 0,Y 384.436,Z 474.818,A -85,B 0,C 180,E1 -12519.995,E2 -12519.995} C_VEL
LIN {X 0,Y 382.194,Z 472.317,A -85,B 0,C 180,E1 -12521.099,E2 -12521.099} C_VEL
LIN {X 0,Y 380.867,Z 470.119,A -85,B 0,C 180,E1 -12521.711,E2 -12521.711} C_VEL
LIN {X 0,Y 378.465,Z 468.621,A -85,B 0,C 180,E1 -12522.671,E2 -12522.671} C_VEL
LIN {X 0,Y 376.7,Z 466.295,A -85,B 0,C 180,E1 -12523.377,E2 -12523.377} C_VEL
LIN {X 0,Y 376.189,Z 464.759,A -85,B 0,C 180,E1 -12523.73,E2 -12523.73} C_VEL
LIN {X 0,Y 376.016,Z 464.174,A -85,B 0,C 180,E1 -12524.338,E2 -12524.338} C_VEL
LIN {X 0,Y 375.996,Z 464.151,A -85,B 0,C 180,E1 -12527.592,E2 -12527.592} C_VEL
LIN {X 0,Y 375.964,Z 464.155,A -85,B 0,C 180,E1 -12530.833,E2 -12530.833} C_VEL
LIN {X 0,Y 375.944,Z 464.158,A -85,B 0,C 180,E1 -12534.285,E2 -12534.285} C_VEL
LIN {X 0,Y 375.902,Z 464.156,A -85,B 0,C 180,E1 -12537.866,E2 -12537.866} C_VEL
LIN {X 0,Y 375.941,Z 464.156,A -85,B 0,C 180,E1 -12541.563,E2 -12541.563} C_VEL
LIN {X 0,Y 375.934,Z 464.135,A -85,B 0,C 180,E1 -12545.418,E2 -12545.418} C_VEL
LIN {X 0,Y 375.918,Z 464.159,A -85,B 0,C 180,E1 -12548.263,E2 -12548.263} C_VEL
LIN {X 0,Y 375.92,Z 464.141,A -85,B 0,C 180,E1 -12550.001,E2 -12550.001} C_VEL
LIN {X 0,Y 375.206,Z 464.218,A -85,B 0,C 180,E1 -12550.895,E2 -12550.895} C_VEL
LIN {X 0,Y 372.318,Z 464.569,A -85,B 0,C 180,E1 -12552.348,E2 -12552.348} C_VEL
LIN {X 0,Y 369.918,Z 464.88,A -85,B 0,C 180,E1 -12553.523,E2 -12553.523} C_VEL
LIN {X 0,Y 368.92,Z 465.017,A -85,B 0,C 180,E1 -12554.432,E2 -12554.432} C_VEL
LIN {X 0,Y 368.854,Z 465.03,A -85,B 0,C 180,E1 -12554.74,E2 -12554.74} C_VEL
LIN {X 0,Y 368.847,Z 465.031,A -85,B 0,C 180,E1 -12558.176,E2 -12558.176} C_VEL
LIN {X 0,Y 368.863,Z 465.035,A -85,B 0,C 180,E1 -12561.368,E2 -12561.368} C_VEL
LIN {X 0,Y 368.919,Z 465.015,A -85,B 0,C 180,E1 -12565.147,E2 -12565.147} C_VEL
LIN {X 0,Y 368.903,Z 465.031,A -85,B 0,C 180,E1 -12569.046,E2 -12569.046} C_VEL
LIN {X 0,Y 368.897,Z 465.019,A -85,B 0,C 180,E1 -12571.559,E2 -12571.559} C_VEL
LIN {X 0,Y 368.889,Z 465.029,A -85,B 0,C 180,E1 -12575.222,E2 -12575.222} C_VEL
LIN {X 0,Y 368.91,Z 465.032,A -85,B 0,C 180,E1 -12577.606,E2 -12577.606} C_VEL
LIN {X 0,Y 368.891,Z 465.008,A -85,B 0,C 180,E1 -12581.104,E2 -12581.104} C_VEL
LIN {X 0,Y 368.926,Z 465.029,A -85,B 0,C 180,E1 -12584.534,E2 -12584.534} C_VEL
LIN {X 0,Y 369.05,Z 465.008,A -85,B 0,C 180,E1 -12586.792,E2 -12586.792} C_VEL
LIN {X 0,Y 369.05,Z 464.988,A -85,B 0,C 180,E1 -12590.133,E2 -12590.133} C_VEL
LIN {X 0,Y 369.148,Z 464.997,A -85,B 0,C 180,E1 -12593.443,E2 -12593.443} C_VEL
LIN {X 0,Y 369.29,Z 464.966,A -85,B 0,C 180,E1 -12597.82,E2 -12597.82} C_VEL
LIN {X 0,Y 369.29,Z 464.977,A -85,B 0,C 180,E1 -12602.183,E2 -12602.183} C_VEL
LIN {X 0,Y 369.151,Z 464.992,A -85,B 0,C 180,E1 -12606.561,E2 -12606.561} C_VEL
LIN {X 0,Y 369.054,Z 464.986,A -85,B 0,C 180,E1 -12609.87,E2 -12609.87} C_VEL
LIN {X 0,Y 368.999,Z 465.02,A -85,B 0,C 180,E1 -12613.75,E2 -12613.75} C_VEL
LIN {X 0,Y 368.935,Z 465.005,A -85,B 0,C 180,E1 -12617.747,E2 -12617.747} C_VEL
LIN {X 0,Y 368.907,Z 465.024,A -85,B 0,C 180,E1 -12621.223,E2 -12621.223} C_VEL
LIN {X 0,Y 368.907,Z 465.029,A -85,B 0,C 180,E1 -12623.875,E2 -12623.875} C_VEL
LIN {X 0,Y 368.857,Z 465.017,A -85,B 0,C 180,E1 -12627.213,E2 -12627.213} C_VEL
LIN {X 0,Y 368.893,Z 465.032,A -85,B 0,C 180,E1 -12629.694,E2 -12629.694} C_VEL
LIN {X 0,Y 368.897,Z 465.022,A -85,B 0,C 180,E1 -12633.044,E2 -12633.044} C_VEL
LIN {X 0,Y 368.911,Z 465.033,A -85,B 0,C 180,E1 -12636.199,E2 -12636.199} C_VEL
LIN {X 0,Y 368.873,Z 465.029,A -85,B 0,C 180,E1 -12638.959,E2 -12638.959} C_VEL
LIN {X 0,Y 368.86,Z 465.041,A -85,B 0,C 180,E1 -12642.006,E2 -12642.006} C_VEL
LIN {X 0,Y 368.872,Z 465.033,A -85,B 0,C 180,E1 -12645.175,E2 -12645.175} C_VEL
LIN {X 0,Y 368.861,Z 465.021,A -85,B 0,C 180,E1 -12648.175,E2 -12648.175} C_VEL
LIN {X 0,Y 368.877,Z 465.035,A -85,B 0,C 180,E1 -12651.368,E2 -12651.368} C_VEL
LIN {X 0,Y 368.933,Z 465.027,A -85,B 0,C 180,E1 -12655.147,E2 -12655.147} C_VEL
LIN {X 0,Y 368.941,Z 465.167,A -85,B 0,C 180,E1 -12658.69,E2 -12658.69} C_VEL
LIN {X 0,Y 370.72,Z 474.144,A -85,B 0,C 180,E1 -12661.71,E2 -12661.71} C_VEL
LIN {X 0,Y 371.975,Z 481.462,A -85,B 0,C 180,E1 -12663.942,E2 -12663.942} C_VEL
LIN {X 0,Y 371.171,Z 490.598,A -85,B 0,C 180,E1 -12666.57,E2 -12666.57} C_VEL
LIN {X 0,Y 370.635,Z 496.495,A -85,B 0,C 180,E1 -12668.27,E2 -12668.27} C_VEL
LIN {X 0,Y 371.515,Z 501.173,A -85,B 0,C 180,E1 -12668.475,E2 -12668.475} C_VEL
LIN {X 0,Y 376.376,Z 527.698,A -85,B 0,C 180,E1 -12669.294,E2 -12669.294} C_VEL
LIN {X 0,Y 376.811,Z 531.855,A -85,B 0,C 180,E1 -12669.401,E2 -12669.401} C_VEL
LIN {X 0,Y 375.721,Z 601.434,A -85,B 0,C 180,E1 -12670.751,E2 -12670.751} C_VEL
LIN {X 0,Y 375.298,Z 611.351,A -85,B 0,C 180,E1 -12671.048,E2 -12671.048} C_VEL
LIN {X 0,Y 374.767,Z 621.34,A -85,B 0,C 180,E1 -12671.481,E2 -12671.481} C_VEL
LIN {X 0,Y 373.931,Z 631.694,A -85,B 0,C 180,E1 -12672.076,E2 -12672.076} C_VEL
LIN {X 0,Y 373.243,Z 640.843,A -85,B 0,C 180,E1 -12672.749,E2 -12672.749} C_VEL
LIN {X 0,Y 372.399,Z 649.845,A -85,B 0,C 180,E1 -12673.556,E2 -12673.556} C_VEL
LIN {X 0,Y 371.569,Z 658.574,A -85,B 0,C 180,E1 -12674.504,E2 -12674.504} C_VEL
LIN {X 0,Y 370.839,Z 666.067,A -85,B 0,C 180,E1 -12675.468,E2 -12675.468} C_VEL
LIN {X 0,Y 369.921,Z 674.795,A -85,B 0,C 180,E1 -12676.822,E2 -12676.822} C_VEL
LIN {X 0,Y 369.259,Z 680.785,A -85,B 0,C 180,E1 -12677.915,E2 -12677.915} C_VEL
LIN {X 0,Y 368.613,Z 687.097,A -85,B 0,C 180,E1 -12679.287,E2 -12679.287} C_VEL
LIN {X 0,Y 368.139,Z 692.372,A -85,B 0,C 180,E1 -12680.661,E2 -12680.661} C_VEL
LIN {X 0,Y 367.734,Z 697.466,A -85,B 0,C 180,E1 -12682.312,E2 -12682.312} C_VEL
LIN {X 0,Y 367.47,Z 701.517,A -85,B 0,C 180,E1 -12684.006,E2 -12684.006} C_VEL
LIN {X 0,Y 367.439,Z 704.365,A -85,B 0,C 180,E1 -12685.612,E2 -12685.612} C_VEL
LIN {X 0,Y 367.38,Z 705.864,A -85,B 0,C 180,E1 -12686.71,E2 -12686.71} C_VEL
LIN {X 0,Y 367.405,Z 707.387,A -85,B 0,C 180,E1 -12688.904,E2 -12688.904} C_VEL
LIN {X 0,Y 367.442,Z 707.667,A -85,B 0,C 180,E1 -12690,E2 -12690} C_VEL
LIN {X 0,Y 367.361,Z 706.791,A -85,B 0,C 180,E1 -12692.193,E2 -12692.193} C_VEL
LIN {X 0,Y 367.38,Z 705.864,A -85,B 0,C 180,E1 -12693.29,E2 -12693.29} C_VEL
LIN {X 0,Y 367.465,Z 702.519,A -85,B 0,C 180,E1 -12695.487,E2 -12695.487} C_VEL
LIN {X 0,Y 367.665,Z 698.894,A -85,B 0,C 180,E1 -12697.137,E2 -12697.137} C_VEL
LIN {X 0,Y 368.005,Z 694.162,A -85,B 0,C 180,E1 -12698.788,E2 -12698.788} C_VEL
LIN {X 0,Y 368.525,Z 688.19,A -85,B 0,C 180,E1 -12700.438,E2 -12700.438} C_VEL
LIN {X 0,Y 369.073,Z 682.096,A -85,B 0,C 180,E1 -12701.812,E2 -12701.812} C_VEL
LIN {X 0,Y 369.743,Z 676.356,A -85,B 0,C 180,E1 -12702.905,E2 -12702.905} C_VEL
LIN {X 0,Y 370.424,Z 669.698,A -85,B 0,C 180,E1 -12703.999,E2 -12703.999} C_VEL
LIN {X 0,Y 371.247,Z 661.794,A -85,B 0,C 180,E1 -12705.097,E2 -12705.097} C_VEL
LIN {X 0,Y 372.002,Z 653.784,A -85,B 0,C 180,E1 -12706.039,E2 -12706.039} C_VEL
LIN {X 0,Y 372.923,Z 644.022,A -85,B 0,C 180,E1 -12706.984,E2 -12706.984} C_VEL
LIN {X 0,Y 373.699,Z 635.633,A -85,B 0,C 180,E1 -12707.653,E2 -12707.653} C_VEL
LIN {X 0,Y 374.475,Z 625.127,A -85,B 0,C 180,E1 -12708.322,E2 -12708.322} C_VEL
LIN {X 0,Y 375.048,Z 614.793,A -85,B 0,C 180,E1 -12708.824,E2 -12708.824} C_VEL
LIN {X 0,Y 375.608,Z 604.077,A -85,B 0,C 180,E1 -12709.184,E2 -12709.184} C_VEL
LIN {X 0,Y 376.111,Z 581.303,A -85,B 0,C 180,E1 -12709.654,E2 -12709.654} C_VEL
LIN {X 0,Y 376.719,Z 529.725,A -85,B 0,C 180,E1 -12710.646,E2 -12710.646} C_VEL
LIN {X 0,Y 371.899,Z 503.021,A -85,B 0,C 180,E1 -12711.464,E2 -12711.464} C_VEL
LIN {X 0,Y 370.619,Z 496.872,A -85,B 0,C 180,E1 -12711.69,E2 -12711.69} C_VEL
LIN {X 0,Y 370.65,Z 495.288,A -85,B 0,C 180,E1 -12712.034,E2 -12712.034} C_VEL
LIN {X 0,Y 371.832,Z 484.517,A -85,B 0,C 180,E1 -12715.212,E2 -12715.212} C_VEL
LIN {X 0,Y 371.88,Z 480.65,A -85,B 0,C 180,E1 -12716.366,E2 -12716.366} C_VEL
LIN {X 0,Y 370.018,Z 470.285,A -85,B 0,C 180,E1 -12719.593,E2 -12719.593} C_VEL
LIN {X 0,Y 368.935,Z 465.131,A -85,B 0,C 180,E1 -12721.351,E2 -12721.351} C_VEL
LIN {X 0,Y 368.926,Z 465.027,A -85,B 0,C 180,E1 -12724.999,E2 -12724.999} C_VEL
LIN {X 0,Y 368.877,Z 465.035,A -85,B 0,C 180,E1 -12728.632,E2 -12728.632} C_VEL
LIN {X 0,Y 368.858,Z 465.022,A -85,B 0,C 180,E1 -12732.004,E2 -12732.004} C_VEL
LIN {X 0,Y 368.873,Z 465.032,A -85,B 0,C 180,E1 -12735.173,E2 -12735.173} C_VEL
LIN {X 0,Y 368.862,Z 465.039,A -85,B 0,C 180,E1 -12738.173,E2 -12738.173} C_VEL
LIN {X 0,Y 368.875,Z 465.029,A -85,B 0,C 180,E1 -12741.365,E2 -12741.365} C_VEL
LIN {X 0,Y 368.931,Z 465.018,A -85,B 0,C 180,E1 -12745.144,E2 -12745.144} C_VEL
LIN {X 0,Y 368.914,Z 465.029,A -85,B 0,C 180,E1 -12749.044,E2 -12749.044} C_VEL
LIN {X 0,Y 368.907,Z 465.026,A -85,B 0,C 180,E1 -12751.556,E2 -12751.556} C_VEL
LIN {X 0,Y 368.885,Z 465.024,A -85,B 0,C 180,E1 -12755.218,E2 -12755.218} C_VEL
LIN {X 0,Y 368.894,Z 465.032,A -85,B 0,C 180,E1 -12757.601,E2 -12757.601} C_VEL
LIN {X 0,Y 368.895,Z 465.008,A -85,B 0,C 180,E1 -12761.101,E2 -12761.101} C_VEL
LIN {X 0,Y 368.918,Z 465.027,A -85,B 0,C 180,E1 -12764.53,E2 -12764.53} C_VEL
LIN {X 0,Y 369.021,Z 465.013,A -85,B 0,C 180,E1 -12766.787,E2 -12766.787} C_VEL
LIN {X 0,Y 369.054,Z 464.986,A -85,B 0,C 180,E1 -12770.13,E2 -12770.13} C_VEL
LIN {X 0,Y 369.151,Z 464.992,A -85,B 0,C 180,E1 -12773.439,E2 -12773.439} C_VEL
LIN {X 0,Y 369.291,Z 464.977,A -85,B 0,C 180,E1 -12777.817,E2 -12777.817} C_VEL
LIN {X 0,Y 369.29,Z 464.966,A -85,B 0,C 180,E1 -12782.18,E2 -12782.18} C_VEL
LIN {X 0,Y 369.148,Z 464.997,A -85,B 0,C 180,E1 -12786.557,E2 -12786.557} C_VEL
LIN {X 0,Y 369.05,Z 464.988,A -85,B 0,C 180,E1 -12789.867,E2 -12789.867} C_VEL
LIN {X 0,Y 369.03,Z 465.014,A -85,B 0,C 180,E1 -12793.77,E2 -12793.77} C_VEL
LIN {X 0,Y 368.928,Z 465.015,A -85,B 0,C 180,E1 -12797.744,E2 -12797.744} C_VEL
LIN {X 0,Y 368.9,Z 465.022,A -85,B 0,C 180,E1 -12801.219,E2 -12801.219} C_VEL
LIN {X 0,Y 368.91,Z 465.034,A -85,B 0,C 180,E1 -12803.876,E2 -12803.876} C_VEL
LIN {X 0,Y 368.847,Z 465.019,A -85,B 0,C 180,E1 -12807.21,E2 -12807.21} C_VEL
LIN {X 0,Y 368.882,Z 465.029,A -85,B 0,C 180,E1 -12809.691,E2 -12809.691} C_VEL
LIN {X 0,Y 368.885,Z 465.028,A -85,B 0,C 180,E1 -12813.041,E2 -12813.041} C_VEL
LIN {X 0,Y 368.899,Z 465.028,A -85,B 0,C 180,E1 -12816.196,E2 -12816.196} C_VEL
LIN {X 0,Y 368.861,Z 465.034,A -85,B 0,C 180,E1 -12818.956,E2 -12818.956} C_VEL
LIN {X 0,Y 368.845,Z 465.033,A -85,B 0,C 180,E1 -12822.004,E2 -12822.004} C_VEL
LIN {X 0,Y 368.859,Z 465.031,A -85,B 0,C 180,E1 -12825.173,E2 -12825.173} C_VEL
LIN {X 0,Y 368.845,Z 465.001,A -85,B 0,C 180,E1 -12828.173,E2 -12828.173} C_VEL
LIN {X 0,Y 368.86,Z 465.036,A -85,B 0,C 180,E1 -12831.366,E2 -12831.366} C_VEL
LIN {X 0,Y 368.916,Z 465.005,A -85,B 0,C 180,E1 -12835.145,E2 -12835.145} C_VEL
LIN {X 0,Y 368.898,Z 465.031,A -85,B 0,C 180,E1 -12839.044,E2 -12839.044} C_VEL
LIN {X 0,Y 368.892,Z 465.021,A -85,B 0,C 180,E1 -12841.557,E2 -12841.557} C_VEL
LIN {X 0,Y 368.883,Z 465.037,A -85,B 0,C 180,E1 -12845.22,E2 -12845.22} C_VEL
LIN {X 0,Y 368.905,Z 465.035,A -85,B 0,C 180,E1 -12847.603,E2 -12847.603} C_VEL
LIN {X 0,Y 368.936,Z 465.031,A -85,B 0,C 180,E1 -12851.105,E2 -12851.105} C_VEL
LIN {X 0,Y 368.956,Z 465.219,A -85,B 0,C 180,E1 -12853.967,E2 -12853.967} C_VEL
LIN {X 0,Y 369.194,Z 466.309,A -85,B 0,C 180,E1 -12854.331,E2 -12854.331} C_VEL
LIN {X 0,Y 370.493,Z 468.667,A -85,B 0,C 180,E1 -12854.81,E2 -12854.81} C_VEL
LIN {X 0,Y 372.876,Z 470.539,A -85,B 0,C 180,E1 -12855.608,E2 -12855.608} C_VEL
LIN {X 0,Y 373.973,Z 471.376,A -85,B 0,C 180,E1 -12855.963,E2 -12855.963} C_VEL
LIN {X 0,Y 375.797,Z 474.304,A -85,B 0,C 180,E1 -12856.692,E2 -12856.692} C_VEL
LIN {X 0,Y 378.432,Z 476.429,A -85,B 0,C 180,E1 -12857.668,E2 -12857.668} C_VEL
LIN {X 0,Y 379.484,Z 477.161,A -85,B 0,C 180,E1 -12858.11,E2 -12858.11} C_VEL
LIN {X 0,Y 381.227,Z 479.777,A -85,B 0,C 180,E1 -12858.906,E2 -12858.906} C_VEL
LIN {X 0,Y 383.696,Z 482.09,A -85,B 0,C 180,E1 -12860.092,E2 -12860.092} C_VEL
LIN {X 0,Y 386.163,Z 483.519,A -85,B 0,C 180,E1 -12861.365,E2 -12861.365} C_VEL
LIN {X 0,Y 388.212,Z 486.533,A -85,B 0,C 180,E1 -12862.72,E2 -12862.72} C_VEL
LIN {X 0,Y 390.281,Z 488.365,A -85,B 0,C 180,E1 -12864.316,E2 -12864.316} C_VEL
LIN {X 0,Y 391.881,Z 489.264,A -85,B 0,C 180,E1 -12865.886,E2 -12865.886} C_VEL
LIN {X 0,Y 392.987,Z 489.664,A -85,B 0,C 180,E1 -12867.454,E2 -12867.454} C_VEL
LIN {X 0,Y 393.531,Z 490.164,A -85,B 0,C 180,E1 -12868.977,E2 -12868.977} C_VEL
LIN {X 0,Y 393.581,Z 490.159,A -85,B 0,C 180,E1 -12870.701,E2 -12870.701} C_VEL
LIN {X 0,Y 393.226,Z 489.787,A -85,B 0,C 180,E1 -12872.048,E2 -12872.048} C_VEL
LIN {X 0,Y 392.186,Z 489.358,A -85,B 0,C 180,E1 -12873.739,E2 -12873.739} C_VEL
LIN {X 0,Y 390.713,Z 488.674,A -85,B 0,C 180,E1 -12875.289,E2 -12875.289} C_VEL
LIN {X 0,Y 388.751,Z 487.139,A -85,B 0,C 180,E1 -12876.879,E2 -12876.879} C_VEL
LIN {X 0,Y 386.961,Z 484.806,A -85,B 0,C 180,E1 -12878.133,E2 -12878.133} C_VEL
LIN {X 0,Y 385.945,Z 483.221,A -85,B 0,C 180,E1 -12878.772,E2 -12878.772} C_VEL
LIN {X 0,Y 383.11,Z 481.666,A -85,B 0,C 180,E1 -12880.192,E2 -12880.192} C_VEL
LIN {X 0,Y 380.722,Z 479.21,A -85,B 0,C 180,E1 -12881.311,E2 -12881.311} C_VEL
LIN {X 0,Y 379.159,Z 476.793,A -85,B 0,C 180,E1 -12882.036,E2 -12882.036} C_VEL
LIN {X 0,Y 376.587,Z 475.13,A -85,B 0,C 180,E1 -12883.004,E2 -12883.004} C_VEL
LIN {X 0,Y 374.521,Z 472.365,A -85,B 0,C 180,E1 -12883.83,E2 -12883.83} C_VEL
LIN {X 0,Y 373.639,Z 470.915,A -85,B 0,C 180,E1 -12884.154,E2 -12884.154} C_VEL
LIN {X 0,Y 370.84,Z 469.032,A -85,B 0,C 180,E1 -12885.069,E2 -12885.069} C_VEL
LIN {X 0,Y 369.417,Z 466.926,A -85,B 0,C 180,E1 -12885.57,E2 -12885.57} C_VEL
LIN {X 0,Y 368.986,Z 465.462,A -85,B 0,C 180,E1 -12885.89,E2 -12885.89} C_VEL
LIN {X 0,Y 368.911,Z 465.034,A -85,B 0,C 180,E1 -12886.604,E2 -12886.604} C_VEL
LIN {X 0,Y 368.913,Z 465.034,A -85,B 0,C 180,E1 -12890.054,E2 -12890.054} C_VEL
LIN {X 0,Y 368.904,Z 465.036,A -85,B 0,C 180,E1 -12893.878,E2 -12893.878} C_VEL
LIN {X 0,Y 368.843,Z 465.041,A -85,B 0,C 180,E1 -12897.213,E2 -12897.213} C_VEL
LIN {X 0,Y 368.877,Z 465.018,A -85,B 0,C 180,E1 -12899.693,E2 -12899.693} C_VEL
LIN {X 0,Y 368.882,Z 465.026,A -85,B 0,C 180,E1 -12903.044,E2 -12903.044} C_VEL
LIN {X 0,Y 368.896,Z 465.021,A -85,B 0,C 180,E1 -12906.199,E2 -12906.199} C_VEL
LIN {X 0,Y 368.847,Z 465.02,A -85,B 0,C 180,E1 -12910.01,E2 -12910.01} C_VEL
LIN {X 0,Y 368.864,Z 465.012,A -85,B 0,C 180,E1 -12913.616,E2 -12913.616} C_VEL
LIN {X 0,Y 368.854,Z 465.03,A -85,B 0,C 180,E1 -12914.74,E2 -12914.74} C_VEL
LIN {X 0,Y 368.224,Z 465.121,A -85,B 0,C 180,E1 -12915.651,E2 -12915.651} C_VEL
LIN {X 0,Y 365.369,Z 465.474,A -85,B 0,C 180,E1 -12917.132,E2 -12917.132} C_VEL
LIN {X 0,Y 362.926,Z 465.767,A -85,B 0,C 180,E1 -12918.331,E2 -12918.331} C_VEL
LIN {X 0,Y 361.874,Z 465.894,A -85,B 0,C 180,E1 -12919.258,E2 -12919.258} C_VEL
LIN {X 0,Y 361.788,Z 465.906,A -85,B 0,C 180,E1 -12919.572,E2 -12919.572} C_VEL
LIN {X 0,Y 361.849,Z 465.909,A -85,B 0,C 180,E1 -12922.983,E2 -12922.983} C_VEL
LIN {X 0,Y 361.847,Z 465.906,A -85,B 0,C 180,E1 -12926.633,E2 -12926.633} C_VEL
LIN {X 0,Y 361.845,Z 465.914,A -85,B 0,C 180,E1 -12929.672,E2 -12929.672} C_VEL
LIN {X 0,Y 361.845,Z 465.893,A -85,B 0,C 180,E1 -12933.469,E2 -12933.469} C_VEL
LIN {X 0,Y 361.866,Z 465.907,A -85,B 0,C 180,E1 -12937.145,E2 -12937.145} C_VEL
LIN {X 0,Y 361.833,Z 465.885,A -85,B 0,C 180,E1 -12940.721,E2 -12940.721} C_VEL
LIN {X 0,Y 361.878,Z 465.909,A -85,B 0,C 180,E1 -12944.225,E2 -12944.225} C_VEL
LIN {X 0,Y 361.992,Z 465.888,A -85,B 0,C 180,E1 -12946.529,E2 -12946.529} C_VEL
LIN {X 0,Y 361.987,Z 465.866,A -85,B 0,C 180,E1 -12949.939,E2 -12949.939} C_VEL
LIN {X 0,Y 362.113,Z 465.873,A -85,B 0,C 180,E1 -12953.315,E2 -12953.315} C_VEL
LIN {X 0,Y 362.252,Z 465.843,A -85,B 0,C 180,E1 -12957.778,E2 -12957.778} C_VEL
LIN {X 0,Y 362.253,Z 465.854,A -85,B 0,C 180,E1 -12962.225,E2 -12962.225} C_VEL
LIN {X 0,Y 362.116,Z 465.868,A -85,B 0,C 180,E1 -12966.689,E2 -12966.689} C_VEL
LIN {X 0,Y 361.99,Z 465.866,A -85,B 0,C 180,E1 -12970.065,E2 -12970.065} C_VEL
LIN {X 0,Y 361.949,Z 465.899,A -85,B 0,C 180,E1 -12973.869,E2 -12973.869} C_VEL
LIN {X 0,Y 361.875,Z 465.881,A -85,B 0,C 180,E1 -12978.105,E2 -12978.105} C_VEL
LIN {X 0,Y 361.851,Z 465.906,A -85,B 0,C 180,E1 -12981.657,E2 -12981.657} C_VEL
LIN {X 0,Y 361.859,Z 465.898,A -85,B 0,C 180,E1 -12985.297,E2 -12985.297} C_VEL
LIN {X 0,Y 361.856,Z 465.905,A -85,B 0,C 180,E1 -12989.075,E2 -12989.075} C_VEL
LIN {X 0,Y 361.848,Z 465.9,A -85,B 0,C 180,E1 -12992.946,E2 -12992.946} C_VEL
LIN {X 0,Y 361.864,Z 465.902,A -85,B 0,C 180,E1 -12995.639,E2 -12995.639} C_VEL
LIN {X 0,Y 361.825,Z 465.907,A -85,B 0,C 180,E1 -12999.019,E2 -12999.019} C_VEL
LIN {X 0,Y 361.83,Z 465.911,A -85,B 0,C 180,E1 -13002.831,E2 -13002.831} C_VEL
LIN {X 0,Y 361.814,Z 465.92,A -85,B 0,C 180,E1 -13005.949,E2 -13005.949} C_VEL
LIN {X 0,Y 361.812,Z 465.893,A -85,B 0,C 180,E1 -13009.251,E2 -13009.251} C_VEL
LIN {X 0,Y 361.863,Z 465.902,A -85,B 0,C 180,E1 -13012.982,E2 -13012.982} C_VEL
LIN {X 0,Y 361.861,Z 465.903,A -85,B 0,C 180,E1 -13016.632,E2 -13016.632} C_VEL
LIN {X 0,Y 361.943,Z 466.108,A -85,B 0,C 180,E1 -13018.381,E2 -13018.381} C_VEL
LIN {X 0,Y 363.476,Z 473.951,A -85,B 0,C 180,E1 -13021.093,E2 -13021.093} C_VEL
LIN {X 0,Y 364.951,Z 482.32,A -85,B 0,C 180,E1 -13023.71,E2 -13023.71} C_VEL
LIN {X 0,Y 364.759,Z 486.473,A -85,B 0,C 180,E1 -13024.92,E2 -13024.92} C_VEL
LIN {X 0,Y 363.725,Z 496.301,A -85,B 0,C 180,E1 -13027.836,E2 -13027.836} C_VEL
LIN {X 0,Y 364.593,Z 500.795,A -85,B 0,C 180,E1 -13028.042,E2 -13028.042} C_VEL
LIN {X 0,Y 369.283,Z 525.517,A -85,B 0,C 180,E1 -13028.837,E2 -13028.837} C_VEL
LIN {X 0,Y 370.155,Z 532.465,A -85,B 0,C 180,E1 -13029.03,E2 -13029.03} C_VEL
LIN {X 0,Y 369.024,Z 601.238,A -85,B 0,C 180,E1 -13030.387,E2 -13030.387} C_VEL
LIN {X 0,Y 368.6,Z 611.156,A -85,B 0,C 180,E1 -13030.69,E2 -13030.69} C_VEL
LIN {X 0,Y 368.056,Z 621.144,A -85,B 0,C 180,E1 -13031.13,E2 -13031.13} C_VEL
LIN {X 0,Y 367.189,Z 631.498,A -85,B 0,C 180,E1 -13031.735,E2 -13031.735} C_VEL
LIN {X 0,Y 366.469,Z 640.646,A -85,B 0,C 180,E1 -13032.42,E2 -13032.42} C_VEL
LIN {X 0,Y 365.584,Z 649.648,A -85,B 0,C 180,E1 -13033.24,E2 -13033.24} C_VEL
LIN {X 0,Y 364.699,Z 658.377,A -85,B 0,C 180,E1 -13034.205,E2 -13034.205} C_VEL
LIN {X 0,Y 363.9,Z 666.256,A -85,B 0,C 180,E1 -13035.244,E2 -13035.244} C_VEL
LIN {X 0,Y 362.977,Z 674.598,A -85,B 0,C 180,E1 -13036.565,E2 -13036.565} C_VEL
LIN {X 0,Y 362.283,Z 680.588,A -85,B 0,C 180,E1 -13037.679,E2 -13037.679} C_VEL
LIN {X 0,Y 361.59,Z 686.899,A -85,B 0,C 180,E1 -13039.076,E2 -13039.076} C_VEL
LIN {X 0,Y 361.089,Z 692.174,A -85,B 0,C 180,E1 -13040.477,E2 -13040.477} C_VEL
LIN {X 0,Y 360.685,Z 697.269,A -85,B 0,C 180,E1 -13042.161,E2 -13042.161} C_VEL
LIN {X 0,Y 360.503,Z 700.109,A -85,B 0,C 180,E1 -13043.283,E2 -13043.283} C_VEL
LIN {X 0,Y 360.35,Z 704.169,A -85,B 0,C 180,E1 -13045.526,E2 -13045.526} C_VEL
LIN {X 0,Y 360.299,Z 705.668,A -85,B 0,C 180,E1 -13046.645,E2 -13046.645} C_VEL
LIN {X 0,Y 360.305,Z 707.191,A -85,B 0,C 180,E1 -13048.882,E2 -13048.882} C_VEL
LIN {X 0,Y 360.344,Z 707.471,A -85,B 0,C 180,E1 -13050,E2 -13050} C_VEL
LIN {X 0,Y 360.266,Z 706.595,A -85,B 0,C 180,E1 -13052.236,E2 -13052.236} C_VEL
LIN {X 0,Y 360.299,Z 705.668,A -85,B 0,C 180,E1 -13053.355,E2 -13053.355} C_VEL
LIN {X 0,Y 360.366,Z 702.322,A -85,B 0,C 180,E1 -13055.596,E2 -13055.596} C_VEL
LIN {X 0,Y 360.598,Z 698.697,A -85,B 0,C 180,E1 -13057.278,E2 -13057.278} C_VEL
LIN {X 0,Y 360.944,Z 693.965,A -85,B 0,C 180,E1 -13058.961,E2 -13058.961} C_VEL
LIN {X 0,Y 361.513,Z 687.993,A -85,B 0,C 180,E1 -13060.643,E2 -13060.643} C_VEL
LIN {X 0,Y 361.948,Z 683.211,A -85,B 0,C 180,E1 -13061.764,E2 -13061.764} C_VEL
LIN {X 0,Y 362.62,Z 677.719,A -85,B 0,C 180,E1 -13062.878,E2 -13062.878} C_VEL
LIN {X 0,Y 363.515,Z 669.501,A -85,B 0,C 180,E1 -13064.27,E2 -13064.27} C_VEL
LIN {X 0,Y 364.288,Z 662.441,A -85,B 0,C 180,E1 -13065.283,E2 -13065.283} C_VEL
LIN {X 0,Y 365.173,Z 653.587,A -85,B 0,C 180,E1 -13066.348,E2 -13066.348} C_VEL
LIN {X 0,Y 366.13,Z 643.826,A -85,B 0,C 180,E1 -13067.309,E2 -13067.309} C_VEL
LIN {X 0,Y 366.939,Z 635.437,A -85,B 0,C 180,E1 -13067.989,E2 -13067.989} C_VEL
LIN {X 0,Y 367.747,Z 624.931,A -85,B 0,C 180,E1 -13068.669,E2 -13068.669} C_VEL
LIN {X 0,Y 368.349,Z 614.597,A -85,B 0,C 180,E1 -13069.179,E2 -13069.179} C_VEL
LIN {X 0,Y 368.926,Z 603.881,A -85,B 0,C 180,E1 -13069.546,E2 -13069.546} C_VEL
LIN {X 0,Y 369.471,Z 579.847,A -85,B 0,C 180,E1 -13070.048,E2 -13070.048} C_VEL
LIN {X 0,Y 370.087,Z 530.504,A -85,B 0,C 180,E1 -13071.014,E2 -13071.014} C_VEL
LIN {X 0,Y 365.174,Z 503.684,A -85,B 0,C 180,E1 -13071.862,E2 -13071.862} C_VEL
LIN {X 0,Y 363.706,Z 496.629,A -85,B 0,C 180,E1 -13072.127,E2 -13072.127} C_VEL
LIN {X 0,Y 363.692,Z 495.921,A -85,B 0,C 180,E1 -13072.238,E2 -13072.238} C_VEL
LIN {X 0,Y 365,Z 484.479,A -85,B 0,C 180,E1 -13075.672,E2 -13075.672} C_VEL
LIN {X 0,Y 364.73,Z 480.603,A -85,B 0,C 180,E1 -13076.877,E2 -13076.877} C_VEL
LIN {X 0,Y 362.743,Z 470.097,A -85,B 0,C 180,E1 -13080.247,E2 -13080.247} C_VEL
LIN {X 0,Y 361.916,Z 465.995,A -85,B 0,C 180,E1 -13081.703,E2 -13081.703} C_VEL
LIN {X 0,Y 361.866,Z 465.898,A -85,B 0,C 180,E1 -13085.636,E2 -13085.636} C_VEL
LIN {X 0,Y 361.827,Z 465.912,A -85,B 0,C 180,E1 -13089.016,E2 -13089.016} C_VEL
LIN {X 0,Y 361.83,Z 465.912,A -85,B 0,C 180,E1 -13092.829,E2 -13092.829} C_VEL
LIN {X 0,Y 361.814,Z 465.91,A -85,B 0,C 180,E1 -13095.947,E2 -13095.947} C_VEL
LIN {X 0,Y 361.811,Z 465.911,A -85,B 0,C 180,E1 -13099.248,E2 -13099.248} C_VEL
LIN {X 0,Y 361.861,Z 465.908,A -85,B 0,C 180,E1 -13102.98,E2 -13102.98} C_VEL
LIN {X 0,Y 361.858,Z 465.896,A -85,B 0,C 180,E1 -13106.63,E2 -13106.63} C_VEL
LIN {X 0,Y 361.856,Z 465.91,A -85,B 0,C 180,E1 -13109.669,E2 -13109.669} C_VEL
LIN {X 0,Y 361.854,Z 465.887,A -85,B 0,C 180,E1 -13113.466,E2 -13113.466} C_VEL
LIN {X 0,Y 361.86,Z 465.906,A -85,B 0,C 180,E1 -13117.141,E2 -13117.141} C_VEL
LIN {X 0,Y 361.837,Z 465.888,A -85,B 0,C 180,E1 -13120.718,E2 -13120.718} C_VEL
LIN {X 0,Y 361.867,Z 465.892,A -85,B 0,C 180,E1 -13123.061,E2 -13123.061} C_VEL
LIN {X 0,Y 361.961,Z 465.893,A -85,B 0,C 180,E1 -13126.525,E2 -13126.525} C_VEL
LIN {X 0,Y 361.99,Z 465.866,A -85,B 0,C 180,E1 -13129.935,E2 -13129.935} C_VEL
LIN {X 0,Y 362.116,Z 465.868,A -85,B 0,C 180,E1 -13133.311,E2 -13133.311} C_VEL
LIN {X 0,Y 362.253,Z 465.854,A -85,B 0,C 180,E1 -13137.775,E2 -13137.775} C_VEL
LIN {X 0,Y 362.252,Z 465.843,A -85,B 0,C 180,E1 -13142.222,E2 -13142.222} C_VEL
LIN {X 0,Y 362.113,Z 465.873,A -85,B 0,C 180,E1 -13146.685,E2 -13146.685} C_VEL
LIN {X 0,Y 361.987,Z 465.866,A -85,B 0,C 180,E1 -13150.061,E2 -13150.061} C_VEL
LIN {X 0,Y 361.973,Z 465.894,A -85,B 0,C 180,E1 -13153.885,E2 -13153.885} C_VEL
LIN {X 0,Y 361.869,Z 465.888,A -85,B 0,C 180,E1 -13158.102,E2 -13158.102} C_VEL
LIN {X 0,Y 361.851,Z 465.902,A -85,B 0,C 180,E1 -13161.653,E2 -13161.653} C_VEL
LIN {X 0,Y 361.856,Z 465.905,A -85,B 0,C 180,E1 -13165.293,E2 -13165.293} C_VEL
LIN {X 0,Y 361.846,Z 465.903,A -85,B 0,C 180,E1 -13169.072,E2 -13169.072} C_VEL
LIN {X 0,Y 361.837,Z 465.906,A -85,B 0,C 180,E1 -13172.943,E2 -13172.943} C_VEL
LIN {X 0,Y 361.852,Z 465.898,A -85,B 0,C 180,E1 -13175.636,E2 -13175.636} C_VEL
LIN {X 0,Y 361.813,Z 465.912,A -85,B 0,C 180,E1 -13179.016,E2 -13179.016} C_VEL
LIN {X 0,Y 361.816,Z 465.914,A -85,B 0,C 180,E1 -13182.829,E2 -13182.829} C_VEL
LIN {X 0,Y 361.799,Z 465.897,A -85,B 0,C 180,E1 -13185.947,E2 -13185.947} C_VEL
LIN {X 0,Y 361.795,Z 465.888,A -85,B 0,C 180,E1 -13189.249,E2 -13189.249} C_VEL
LIN {X 0,Y 361.846,Z 465.909,A -85,B 0,C 180,E1 -13192.98,E2 -13192.98} C_VEL
LIN {X 0,Y 361.843,Z 465.896,A -85,B 0,C 180,E1 -13196.63,E2 -13196.63} C_VEL
LIN {X 0,Y 361.841,Z 465.901,A -85,B 0,C 180,E1 -13199.669,E2 -13199.669} C_VEL
LIN {X 0,Y 361.84,Z 465.914,A -85,B 0,C 180,E1 -13203.466,E2 -13203.466} C_VEL
LIN {X 0,Y 361.861,Z 465.912,A -85,B 0,C 180,E1 -13207.143,E2 -13207.143} C_VEL
LIN {X 0,Y 361.866,Z 465.912,A -85,B 0,C 180,E1 -13210.721,E2 -13210.721} C_VEL
LIN {X 0,Y 361.949,Z 466.169,A -85,B 0,C 180,E1 -13212.255,E2 -13212.255} C_VEL
LIN {X 0,Y 362.231,Z 467.371,A -85,B 0,C 180,E1 -13212.565,E2 -13212.565} C_VEL
LIN {X 0,Y 363.754,Z 469.912,A -85,B 0,C 180,E1 -13213.046,E2 -13213.046} C_VEL
LIN {X 0,Y 366.347,Z 471.948,A -85,B 0,C 180,E1 -13213.812,E2 -13213.812} C_VEL
LIN {X 0,Y 368.225,Z 474.917,A -85,B 0,C 180,E1 -13214.424,E2 -13214.424} C_VEL
LIN {X 0,Y 370.683,Z 476.99,A -85,B 0,C 180,E1 -13215.216,E2 -13215.216} C_VEL
LIN {X 0,Y 371.959,Z 478.031,A -85,B 0,C 180,E1 -13215.641,E2 -13215.641} C_VEL
LIN {X 0,Y 374.183,Z 481.049,A -85,B 0,C 180,E1 -13216.448,E2 -13216.448} C_VEL
LIN {X 0,Y 376.963,Z 483.266,A -85,B 0,C 180,E1 -13217.483,E2 -13217.483} C_VEL
LIN {X 0,Y 377.846,Z 483.94,A -85,B 0,C 180,E1 -13217.819,E2 -13217.819} C_VEL
LIN {X 0,Y 380.015,Z 486.89,A -85,B 0,C 180,E1 -13218.803,E2 -13218.803} C_VEL
LIN {X 0,Y 382.487,Z 489.022,A -85,B 0,C 180,E1 -13219.953,E2 -13219.953} C_VEL
LIN {X 0,Y 384.871,Z 490.359,A -85,B 0,C 180,E1 -13221.137,E2 -13221.137} C_VEL
LIN {X 0,Y 387.159,Z 493.524,A -85,B 0,C 180,E1 -13222.601,E2 -13222.601} C_VEL
LIN {X 0,Y 389.389,Z 495.431,A -85,B 0,C 180,E1 -13224.303,E2 -13224.303} C_VEL
LIN {X 0,Y 391.006,Z 496.311,A -85,B 0,C 180,E1 -13225.877,E2 -13225.877} C_VEL
LIN {X 0,Y 392.12,Z 496.712,A -85,B 0,C 180,E1 -13227.448,E2 -13227.448} C_VEL
LIN {X 0,Y 392.669,Z 497.211,A -85,B 0,C 180,E1 -13228.974,E2 -13228.974} C_VEL
LIN {X 0,Y 392.841,Z 497.213,A -85,B 0,C 180,E1 -13230,E2 -13230} C_VEL
LIN {X 0,Y 392.5,Z 496.947,A -85,B 0,C 180,E1 -13231.779,E2 -13231.779} C_VEL
LIN {X 0,Y 391.86,Z 496.571,A -85,B 0,C 180,E1 -13233.084,E2 -13233.084} C_VEL
LIN {X 0,Y 390.277,Z 495.995,A -85,B 0,C 180,E1 -13234.907,E2 -13234.907} C_VEL
LIN {X 0,Y 388.205,Z 494.524,A -85,B 0,C 180,E1 -13236.637,E2 -13236.637} C_VEL
LIN {X 0,Y 386.251,Z 492.422,A -85,B 0,C 180,E1 -13238,E2 -13238} C_VEL
LIN {X 0,Y 384.53,Z 490.044,A -85,B 0,C 180,E1 -13239.07,E2 -13239.07} C_VEL
LIN {X 0,Y 381.45,Z 488.202,A -85,B 0,C 180,E1 -13240.563,E2 -13240.563} C_VEL
LIN {X 0,Y 378.699,Z 485.316,A -85,B 0,C 180,E1 -13241.779,E2 -13241.779} C_VEL
LIN {X 0,Y 377.389,Z 483.461,A -85,B 0,C 180,E1 -13242.366,E2 -13242.366} C_VEL
LIN {X 0,Y 374.645,Z 481.528,A -85,B 0,C 180,E1 -13243.372,E2 -13243.372} C_VEL
LIN {X 0,Y 372.335,Z 478.645,A -85,B 0,C 180,E1 -13244.223,E2 -13244.223} C_VEL
LIN {X 0,Y 371.41,Z 477.413,A -85,B 0,C 180,E1 -13244.548,E2 -13244.548} C_VEL
LIN {X 0,Y 368.741,Z 475.427,A -85,B 0,C 180,E1 -13245.422,E2 -13245.422} C_VEL
LIN {X 0,Y 366.834,Z 472.872,A -85,B 0,C 180,E1 -13246.022,E2 -13246.022} C_VEL
LIN {X 0,Y 366.062,Z 471.572,A -85,B 0,C 180,E1 -13246.28,E2 -13246.28} C_VEL
LIN {X 0,Y 363.658,Z 469.784,A -85,B 0,C 180,E1 -13246.981,E2 -13246.981} C_VEL
LIN {X 0,Y 362.143,Z 467.103,A -85,B 0,C 180,E1 -13247.482,E2 -13247.482} C_VEL
LIN {X 0,Y 361.967,Z 466.128,A -85,B 0,C 180,E1 -13247.766,E2 -13247.766} C_VEL
LIN {X 0,Y 361.845,Z 465.914,A -85,B 0,C 180,E1 -13251.656,E2 -13251.656} C_VEL
LIN {X 0,Y 361.851,Z 465.913,A -85,B 0,C 180,E1 -13255.296,E2 -13255.296} C_VEL
LIN {X 0,Y 361.841,Z 465.894,A -85,B 0,C 180,E1 -13259.075,E2 -13259.075} C_VEL
LIN {X 0,Y 361.833,Z 465.905,A -85,B 0,C 180,E1 -13262.946,E2 -13262.946} C_VEL
LIN {X 0,Y 361.849,Z 465.89,A -85,B 0,C 180,E1 -13265.638,E2 -13265.638} C_VEL
LIN {X 0,Y 361.81,Z 465.913,A -85,B 0,C 180,E1 -13269.019,E2 -13269.019} C_VEL
LIN {X 0,Y 361.815,Z 465.879,A -85,B 0,C 180,E1 -13272.831,E2 -13272.831} C_VEL
LIN {X 0,Y 361.8,Z 465.917,A -85,B 0,C 180,E1 -13275.949,E2 -13275.949} C_VEL
LIN {X 0,Y 361.788,Z 465.906,A -85,B 0,C 180,E1 -13279.572,E2 -13279.572} C_VEL
LIN {X 0,Y 361.13,Z 465.997,A -85,B 0,C 180,E1 -13280.501,E2 -13280.501} C_VEL
LIN {X 0,Y 358.313,Z 466.356,A -85,B 0,C 180,E1 -13282.013,E2 -13282.013} C_VEL
LIN {X 0,Y 355.922,Z 466.648,A -85,B 0,C 180,E1 -13283.236,E2 -13283.236} C_VEL
LIN {X 0,Y 354.887,Z 466.767,A -85,B 0,C 180,E1 -13284.182,E2 -13284.182} C_VEL
LIN {X 0,Y 354.798,Z 466.775,A -85,B 0,C 180,E1 -13284.502,E2 -13284.502} C_VEL
LIN {X 0,Y 354.776,Z 466.789,A -85,B 0,C 180,E1 -13287.668,E2 -13287.668} C_VEL
LIN {X 0,Y 354.779,Z 466.776,A -85,B 0,C 180,E1 -13291.615,E2 -13291.615} C_VEL
LIN {X 0,Y 354.796,Z 466.786,A -85,B 0,C 180,E1 -13295.421,E2 -13295.421} C_VEL
LIN {X 0,Y 354.81,Z 466.777,A -85,B 0,C 180,E1 -13299.114,E2 -13299.114} C_VEL
LIN {X 0,Y 354.83,Z 466.777,A -85,B 0,C 180,E1 -13302.719,E2 -13302.719} C_VEL
LIN {X 0,Y 354.932,Z 466.769,A -85,B 0,C 180,E1 -13306.256,E2 -13306.256} C_VEL
LIN {X 0,Y 354.943,Z 466.743,A -85,B 0,C 180,E1 -13309.737,E2 -13309.737} C_VEL
LIN {X 0,Y 355.079,Z 466.749,A -85,B 0,C 180,E1 -13313.181,E2 -13313.181} C_VEL
LIN {X 0,Y 355.214,Z 466.72,A -85,B 0,C 180,E1 -13317.734,E2 -13317.734} C_VEL
LIN {X 0,Y 355.14,Z 466.728,A -85,B 0,C 180,E1 -13321.136,E2 -13321.136} C_VEL
LIN {X 0,Y 355.215,Z 466.73,A -85,B 0,C 180,E1 -13322.27,E2 -13322.27} C_VEL
LIN {X 0,Y 355.083,Z 466.743,A -85,B 0,C 180,E1 -13326.822,E2 -13326.822} C_VEL
LIN {X 0,Y 354.946,Z 466.745,A -85,B 0,C 180,E1 -13330.267,E2 -13330.267} C_VEL
LIN {X 0,Y 354.89,Z 466.778,A -85,B 0,C 180,E1 -13333.987,E2 -13333.987} C_VEL
LIN {X 0,Y 354.833,Z 466.757,A -85,B 0,C 180,E1 -13338.066,E2 -13338.066} C_VEL
LIN {X 0,Y 354.804,Z 466.789,A -85,B 0,C 180,E1 -13342.11,E2 -13342.11} C_VEL
LIN {X 0,Y 354.799,Z 466.769,A -85,B 0,C 180,E1 -13345.837,E2 -13345.837} C_VEL
LIN {X 0,Y 354.797,Z 466.788,A -85,B 0,C 180,E1 -13349.685,E2 -13349.685} C_VEL
LIN {X 0,Y 354.787,Z 466.781,A -85,B 0,C 180,E1 -13352.335,E2 -13352.335} C_VEL
LIN {X 0,Y 354.819,Z 466.78,A -85,B 0,C 180,E1 -13355.699,E2 -13355.699} C_VEL
LIN {X 0,Y 354.77,Z 466.784,A -85,B 0,C 180,E1 -13359.414,E2 -13359.414} C_VEL
LIN {X 0,Y 354.783,Z 466.789,A -85,B 0,C 180,E1 -13362.867,E2 -13362.867} C_VEL
LIN {X 0,Y 354.763,Z 466.796,A -85,B 0,C 180,E1 -13366.104,E2 -13366.104} C_VEL
LIN {X 0,Y 354.764,Z 466.77,A -85,B 0,C 180,E1 -13369.176,E2 -13369.176} C_VEL
LIN {X 0,Y 354.801,Z 466.787,A -85,B 0,C 180,E1 -13372.406,E2 -13372.406} C_VEL
LIN {X 0,Y 354.81,Z 466.782,A -85,B 0,C 180,E1 -13374.941,E2 -13374.941} C_VEL
LIN {X 0,Y 354.863,Z 466.899,A -85,B 0,C 180,E1 -13377.976,E2 -13377.976} C_VEL
LIN {X 0,Y 356.423,Z 474.805,A -85,B 0,C 180,E1 -13380.79,E2 -13380.79} C_VEL
LIN {X 0,Y 357.917,Z 483.177,A -85,B 0,C 180,E1 -13383.467,E2 -13383.467} C_VEL
LIN {X 0,Y 357.887,Z 486.906,A -85,B 0,C 180,E1 -13384.601,E2 -13384.601} C_VEL
LIN {X 0,Y 356.848,Z 496.095,A -85,B 0,C 180,E1 -13387.384,E2 -13387.384} C_VEL
LIN {X 0,Y 357.778,Z 500.849,A -85,B 0,C 180,E1 -13387.606,E2 -13387.606} C_VEL
LIN {X 0,Y 361.956,Z 522.59,A -85,B 0,C 180,E1 -13388.331,E2 -13388.331} C_VEL
LIN {X 0,Y 363.505,Z 532.203,A -85,B 0,C 180,E1 -13388.627,E2 -13388.627} C_VEL
LIN {X 0,Y 362.355,Z 601.045,A -85,B 0,C 180,E1 -13390.011,E2 -13390.011} C_VEL
LIN {X 0,Y 361.887,Z 610.959,A -85,B 0,C 180,E1 -13390.317,E2 -13390.317} C_VEL
LIN {X 0,Y 361.357,Z 620.949,A -85,B 0,C 180,E1 -13390.767,E2 -13390.767} C_VEL
LIN {X 0,Y 360.468,Z 631.303,A -85,B 0,C 180,E1 -13391.382,E2 -13391.382} C_VEL
LIN {X 0,Y 359.688,Z 640.45,A -85,B 0,C 180,E1 -13392.077,E2 -13392.077} C_VEL
LIN {X 0,Y 358.751,Z 649.451,A -85,B 0,C 180,E1 -13392.911,E2 -13392.911} C_VEL
LIN {X 0,Y 357.835,Z 658.18,A -85,B 0,C 180,E1 -13393.894,E2 -13393.894} C_VEL
LIN {X 0,Y 356.967,Z 666.417,A -85,B 0,C 180,E1 -13395.007,E2 -13395.007} C_VEL
LIN {X 0,Y 356.042,Z 674.401,A -85,B 0,C 180,E1 -13396.298,E2 -13396.298} C_VEL
LIN {X 0,Y 355.326,Z 680.391,A -85,B 0,C 180,E1 -13397.434,E2 -13397.434} C_VEL
LIN {X 0,Y 354.583,Z 686.702,A -85,B 0,C 180,E1 -13398.858,E2 -13398.858} C_VEL
LIN {X 0,Y 354.054,Z 691.977,A -85,B 0,C 180,E1 -13400.286,E2 -13400.286} C_VEL
LIN {X 0,Y 353.628,Z 697.072,A -85,B 0,C 180,E1 -13402.003,E2 -13402.003} C_VEL
LIN {X 0,Y 353.422,Z 699.912,A -85,B 0,C 180,E1 -13403.148,E2 -13403.148} C_VEL
LIN {X 0,Y 353.263,Z 703.972,A -85,B 0,C 180,E1 -13405.436,E2 -13405.436} C_VEL
LIN {X 0,Y 353.221,Z 705.472,A -85,B 0,C 180,E1 -13406.578,E2 -13406.578} C_VEL
LIN {X 0,Y 353.205,Z 706.994,A -85,B 0,C 180,E1 -13408.86,E2 -13408.86} C_VEL
LIN {X 0,Y 353.247,Z 707.274,A -85,B 0,C 180,E1 -13410,E2 -13410} C_VEL
LIN {X 0,Y 353.174,Z 706.398,A -85,B 0,C 180,E1 -13412.281,E2 -13412.281} C_VEL
LIN {X 0,Y 353.221,Z 705.472,A -85,B 0,C 180,E1 -13413.422,E2 -13413.422} C_VEL
LIN {X 0,Y 353.286,Z 702.125,A -85,B 0,C 180,E1 -13415.708,E2 -13415.708} C_VEL
LIN {X 0,Y 353.522,Z 698.5,A -85,B 0,C 180,E1 -13417.424,E2 -13417.424} C_VEL
LIN {X 0,Y 353.9,Z 693.768,A -85,B 0,C 180,E1 -13419.141,E2 -13419.141} C_VEL
LIN {X 0,Y 354.479,Z 687.795,A -85,B 0,C 180,E1 -13420.856,E2 -13420.856} C_VEL
LIN {X 0,Y 355.149,Z 681.702,A -85,B 0,C 180,E1 -13422.282,E2 -13422.282} C_VEL
LIN {X 0,Y 355.866,Z 675.962,A -85,B 0,C 180,E1 -13423.418,E2 -13423.418} C_VEL
LIN {X 0,Y 356.626,Z 669.305,A -85,B 0,C 180,E1 -13424.552,E2 -13424.552} C_VEL
LIN {X 0,Y 357.528,Z 661.163,A -85,B 0,C 180,E1 -13425.723,E2 -13425.723} C_VEL
LIN {X 0,Y 358.347,Z 653.391,A -85,B 0,C 180,E1 -13426.668,E2 -13426.668} C_VEL
LIN {X 0,Y 359.334,Z 643.629,A -85,B 0,C 180,E1 -13427.647,E2 -13427.647} C_VEL
LIN {X 0,Y 360.187,Z 635.241,A -85,B 0,C 180,E1 -13428.338,E2 -13428.338} C_VEL
LIN {X 0,Y 361.035,Z 624.735,A -85,B 0,C 180,E1 -13429.03,E2 -13429.03} C_VEL
LIN {X 0,Y 361.627,Z 614.4,A -85,B 0,C 180,E1 -13429.55,E2 -13429.55} C_VEL
LIN {X 0,Y 362.248,Z 603.685,A -85,B 0,C 180,E1 -13429.921,E2 -13429.921} C_VEL
LIN {X 0,Y 362.792,Z 579.73,A -85,B 0,C 180,E1 -13430.432,E2 -13430.432} C_VEL
LIN {X 0,Y 363.404,Z 531.204,A -85,B 0,C 180,E1 -13431.4,E2 -13431.4} C_VEL
LIN {X 0,Y 358.831,Z 505.903,A -85,B 0,C 180,E1 -13432.218,E2 -13432.218} C_VEL
LIN {X 0,Y 356.832,Z 496.289,A -85,B 0,C 180,E1 -13432.59,E2 -13432.59} C_VEL
LIN {X 0,Y 356.992,Z 494.077,A -85,B 0,C 180,E1 -13433.187,E2 -13433.187} C_VEL
LIN {X 0,Y 358.089,Z 484.283,A -85,B 0,C 180,E1 -13436.205,E2 -13436.205} C_VEL
LIN {X 0,Y 356.713,Z 476.163,A -85,B 0,C 180,E1 -13438.862,E2 -13438.862} C_VEL
LIN {X 0,Y 354.864,Z 466.886,A -85,B 0,C 180,E1 -13442.024,E2 -13442.024} C_VEL
LIN {X 0,Y 354.821,Z 466.775,A -85,B 0,C 180,E1 -13445.697,E2 -13445.697} C_VEL
LIN {X 0,Y 354.771,Z 466.783,A -85,B 0,C 180,E1 -13449.411,E2 -13449.411} C_VEL
LIN {X 0,Y 354.782,Z 466.789,A -85,B 0,C 180,E1 -13452.864,E2 -13452.864} C_VEL
LIN {X 0,Y 354.763,Z 466.788,A -85,B 0,C 180,E1 -13456.101,E2 -13456.101} C_VEL
LIN {X 0,Y 354.764,Z 466.789,A -85,B 0,C 180,E1 -13459.174,E2 -13459.174} C_VEL
LIN {X 0,Y 354.799,Z 466.791,A -85,B 0,C 180,E1 -13462.404,E2 -13462.404} C_VEL
LIN {X 0,Y 354.809,Z 466.778,A -85,B 0,C 180,E1 -13464.939,E2 -13464.939} C_VEL
LIN {X 0,Y 354.794,Z 466.79,A -85,B 0,C 180,E1 -13468.404,E2 -13468.404} C_VEL
LIN {X 0,Y 354.797,Z 466.781,A -85,B 0,C 180,E1 -13471.613,E2 -13471.613} C_VEL
LIN {X 0,Y 354.804,Z 466.779,A -85,B 0,C 180,E1 -13475.418,E2 -13475.418} C_VEL
LIN {X 0,Y 354.816,Z 466.779,A -85,B 0,C 180,E1 -13479.111,E2 -13479.111} C_VEL
LIN {X 0,Y 354.835,Z 466.765,A -85,B 0,C 180,E1 -13482.715,E2 -13482.715} C_VEL
LIN {X 0,Y 354.906,Z 466.775,A -85,B 0,C 180,E1 -13486.252,E2 -13486.252} C_VEL
LIN {X 0,Y 354.946,Z 466.745,A -85,B 0,C 180,E1 -13489.733,E2 -13489.733} C_VEL
LIN {X 0,Y 355.083,Z 466.743,A -85,B 0,C 180,E1 -13493.178,E2 -13493.178} C_VEL
LIN {X 0,Y 355.215,Z 466.73,A -85,B 0,C 180,E1 -13497.73,E2 -13497.73} C_VEL
LIN {X 0,Y 355.139,Z 466.719,A -85,B 0,C 180,E1 -13501.132,E2 -13501.132} C_VEL
LIN {X 0,Y 355.214,Z 466.72,A -85,B 0,C 180,E1 -13502.266,E2 -13502.266} C_VEL
LIN {X 0,Y 355.079,Z 466.749,A -85,B 0,C 180,E1 -13506.819,E2 -13506.819} C_VEL
LIN {X 0,Y 354.943,Z 466.743,A -85,B 0,C 180,E1 -13510.263,E2 -13510.263} C_VEL
LIN {X 0,Y 354.916,Z 466.774,A -85,B 0,C 180,E1 -13514.004,E2 -13514.004} C_VEL
LIN {X 0,Y 354.827,Z 466.765,A -85,B 0,C 180,E1 -13518.063,E2 -13518.063} C_VEL
LIN {X 0,Y 354.805,Z 466.785,A -85,B 0,C 180,E1 -13522.106,E2 -13522.106} C_VEL
LIN {X 0,Y 354.792,Z 466.779,A -85,B 0,C 180,E1 -13525.833,E2 -13525.833} C_VEL
LIN {X 0,Y 354.786,Z 466.785,A -85,B 0,C 180,E1 -13529.682,E2 -13529.682} C_VEL
LIN {X 0,Y 354.776,Z 466.789,A -85,B 0,C 180,E1 -13532.332,E2 -13532.332} C_VEL
LIN {X 0,Y 354.806,Z 466.776,A -85,B 0,C 180,E1 -13535.697,E2 -13535.697} C_VEL
LIN {X 0,Y 354.756,Z 466.792,A -85,B 0,C 180,E1 -13539.411,E2 -13539.411} C_VEL
LIN {X 0,Y 354.768,Z 466.792,A -85,B 0,C 180,E1 -13542.864,E2 -13542.864} C_VEL
LIN {X 0,Y 354.748,Z 466.772,A -85,B 0,C 180,E1 -13546.101,E2 -13546.101} C_VEL
LIN {X 0,Y 354.748,Z 466.763,A -85,B 0,C 180,E1 -13549.174,E2 -13549.174} C_VEL
LIN {X 0,Y 354.784,Z 466.792,A -85,B 0,C 180,E1 -13552.404,E2 -13552.404} C_VEL
LIN {X 0,Y 354.793,Z 466.763,A -85,B 0,C 180,E1 -13554.939,E2 -13554.939} C_VEL
LIN {X 0,Y 354.779,Z 466.793,A -85,B 0,C 180,E1 -13558.404,E2 -13558.404} C_VEL
LIN {X 0,Y 354.774,Z 466.779,A -85,B 0,C 180,E1 -13561.613,E2 -13561.613} C_VEL
LIN {X 0,Y 354.791,Z 466.793,A -85,B 0,C 180,E1 -13565.419,E2 -13565.419} C_VEL
LIN {X 0,Y 354.81,Z 466.79,A -85,B 0,C 180,E1 -13569.112,E2 -13569.112} C_VEL
LIN {X 0,Y 354.869,Z 467.047,A -85,B 0,C 180,E1 -13570.664,E2 -13570.664} C_VEL
LIN {X 0,Y 355.2,Z 468.328,A -85,B 0,C 180,E1 -13570.968,E2 -13570.968} C_VEL
LIN {X 0,Y 356.787,Z 470.871,A -85,B 0,C 180,E1 -13571.426,E2 -13571.426} C_VEL
LIN {X 0,Y 359.098,Z 472.727,A -85,B 0,C 180,E1 -13572.017,E2 -13572.017} C_VEL
LIN {X 0,Y 361.053,Z 475.855,A -85,B 0,C 180,E1 -13572.608,E2 -13572.608} C_VEL
LIN {X 0,Y 364.097,Z 478.552,A -85,B 0,C 180,E1 -13573.451,E2 -13573.451} C_VEL
LIN {X 0,Y 366.37,Z 481.657,A -85,B 0,C 180,E1 -13574.186,E2 -13574.186} C_VEL
LIN {X 0,Y 369.265,Z 483.886,A -85,B 0,C 180,E1 -13575.072,E2 -13575.072} C_VEL
LIN {X 0,Y 370.679,Z 485.669,A -85,B 0,C 180,E1 -13575.573,E2 -13575.573} C_VEL
LIN {X 0,Y 373.488,Z 488.699,A -85,B 0,C 180,E1 -13576.561,E2 -13576.561} C_VEL
LIN {X 0,Y 376.186,Z 490.769,A -85,B 0,C 180,E1 -13577.559,E2 -13577.559} C_VEL
LIN {X 0,Y 378.772,Z 493.918,A -85,B 0,C 180,E1 -13578.683,E2 -13578.683} C_VEL
LIN {X 0,Y 381.162,Z 495.877,A -85,B 0,C 180,E1 -13579.755,E2 -13579.755} C_VEL
LIN {X 0,Y 383.564,Z 497.228,A -85,B 0,C 180,E1 -13580.907,E2 -13580.907} C_VEL
LIN {X 0,Y 386.09,Z 500.505,A -85,B 0,C 180,E1 -13582.481,E2 -13582.481} C_VEL
LIN {X 0,Y 388.469,Z 502.475,A -85,B 0,C 180,E1 -13584.264,E2 -13584.264} C_VEL
LIN {X 0,Y 390.133,Z 503.343,A -85,B 0,C 180,E1 -13585.868,E2 -13585.868} C_VEL
LIN {X 0,Y 391.254,Z 503.761,A -85,B 0,C 180,E1 -13587.443,E2 -13587.443} C_VEL
LIN {X 0,Y 391.81,Z 504.232,A -85,B 0,C 180,E1 -13588.972,E2 -13588.972} C_VEL
LIN {X 0,Y 391.976,Z 504.259,A -85,B 0,C 180,E1 -13590,E2 -13590} C_VEL
LIN {X 0,Y 391.635,Z 503.981,A -85,B 0,C 180,E1 -13591.783,E2 -13591.783} C_VEL
LIN {X 0,Y 390.439,Z 503.424,A -85,B 0,C 180,E1 -13593.756,E2 -13593.756} C_VEL
LIN {X 0,Y 389.079,Z 502.879,A -85,B 0,C 180,E1 -13595.182,E2 -13595.182} C_VEL
LIN {X 0,Y 387.142,Z 501.472,A -85,B 0,C 180,E1 -13596.758,E2 -13596.758} C_VEL
LIN {X 0,Y 385.294,Z 499.633,A -85,B 0,C 180,E1 -13598.02,E2 -13598.02} C_VEL
LIN {X 0,Y 383.254,Z 496.935,A -85,B 0,C 180,E1 -13599.261,E2 -13599.261} C_VEL
LIN {X 0,Y 380.182,Z 495.095,A -85,B 0,C 180,E1 -13600.72,E2 -13600.72} C_VEL
LIN {X 0,Y 377.159,Z 492.098,A -85,B 0,C 180,E1 -13602.032,E2 -13602.032} C_VEL
LIN {X 0,Y 375.477,Z 490.078,A -85,B 0,C 180,E1 -13602.705,E2 -13602.705} C_VEL
LIN {X 0,Y 372.557,Z 487.823,A -85,B 0,C 180,E1 -13603.78,E2 -13603.78} C_VEL
LIN {X 0,Y 369.913,Z 484.549,A -85,B 0,C 180,E1 -13604.704,E2 -13604.704} C_VEL
LIN {X 0,Y 366.109,Z 481.393,A -85,B 0,C 180,E1 -13605.894,E2 -13605.894} C_VEL
LIN {X 0,Y 363.945,Z 478.218,A -85,B 0,C 180,E1 -13606.603,E2 -13606.603} C_VEL
LIN {X 0,Y 360.924,Z 475.722,A -85,B 0,C 180,E1 -13607.428,E2 -13607.428} C_VEL
LIN {X 0,Y 358.698,Z 472.254,A -85,B 0,C 180,E1 -13608.1,E2 -13608.1} C_VEL
LIN {X 0,Y 356.336,Z 470.365,A -85,B 0,C 180,E1 -13608.689,E2 -13608.689} C_VEL
LIN {X 0,Y 354.953,Z 467.474,A -85,B 0,C 180,E1 -13609.181,E2 -13609.181} C_VEL
LIN {X 0,Y 354.816,Z 466.843,A -85,B 0,C 180,E1 -13609.527,E2 -13609.527} C_VEL
LIN {X 0,Y 354.795,Z 466.793,A -85,B 0,C 180,E1 -13613.339,E2 -13613.339} C_VEL
LIN {X 0,Y 354.779,Z 466.793,A -85,B 0,C 180,E1 -13617.104,E2 -13617.104} C_VEL
LIN {X 0,Y 354.782,Z 466.773,A -85,B 0,C 180,E1 -13619.685,E2 -13619.685} C_VEL
LIN {X 0,Y 354.772,Z 466.791,A -85,B 0,C 180,E1 -13622.334,E2 -13622.334} C_VEL
LIN {X 0,Y 354.803,Z 466.768,A -85,B 0,C 180,E1 -13625.699,E2 -13625.699} C_VEL
LIN {X 0,Y 354.755,Z 466.786,A -85,B 0,C 180,E1 -13629.414,E2 -13629.414} C_VEL
LIN {X 0,Y 354.767,Z 466.756,A -85,B 0,C 180,E1 -13632.867,E2 -13632.867} C_VEL
LIN {X 0,Y 354.749,Z 466.797,A -85,B 0,C 180,E1 -13636.104,E2 -13636.104} C_VEL
LIN {X 0,Y 354.73,Z 466.784,A -85,B 0,C 180,E1 -13639.567,E2 -13639.567} C_VEL
LIN {X 0,Y 354.787,Z 466.791,A -85,B 0,C 180,E1 -13642.406,E2 -13642.406} C_VEL
LIN {X 0,Y 354.798,Z 466.775,A -85,B 0,C 180,E1 -13644.502,E2 -13644.502} C_VEL
LIN {X 0,Y 354.108,Z 466.86,A -85,B 0,C 180,E1 -13645.449,E2 -13645.449} C_VEL
LIN {X 0,Y 351.215,Z 467.229,A -85,B 0,C 180,E1 -13646.989,E2 -13646.989} C_VEL
LIN {X 0,Y 348.794,Z 467.54,A -85,B 0,C 180,E1 -13648.235,E2 -13648.235} C_VEL
LIN {X 0,Y 347.786,Z 467.663,A -85,B 0,C 180,E1 -13649.199,E2 -13649.199} C_VEL
LIN {X 0,Y 347.72,Z 467.672,A -85,B 0,C 180,E1 -13649.526,E2 -13649.526} C_VEL
LIN {X 0,Y 347.738,Z 467.646,A -85,B 0,C 180,E1 -13652.78,E2 -13652.78} C_VEL
LIN {X 0,Y 347.743,Z 467.67,A -85,B 0,C 180,E1 -13656.161,E2 -13656.161} C_VEL
LIN {X 0,Y 347.77,Z 467.654,A -85,B 0,C 180,E1 -13658.671,E2 -13658.671} C_VEL
LIN {X 0,Y 347.79,Z 467.647,A -85,B 0,C 180,E1 -13662.357,E2 -13662.357} C_VEL
LIN {X 0,Y 347.892,Z 467.649,A -85,B 0,C 180,E1 -13665.973,E2 -13665.973} C_VEL
LIN {X 0,Y 347.883,Z 467.622,A -85,B 0,C 180,E1 -13669.526,E2 -13669.526} C_VEL
LIN {X 0,Y 348.046,Z 467.624,A -85,B 0,C 180,E1 -13673.043,E2 -13673.043} C_VEL
LIN {X 0,Y 348.175,Z 467.596,A -85,B 0,C 180,E1 -13677.688,E2 -13677.688} C_VEL
LIN {X 0,Y 348.111,Z 467.603,A -85,B 0,C 180,E1 -13681.159,E2 -13681.159} C_VEL
LIN {X 0,Y 348.176,Z 467.607,A -85,B 0,C 180,E1 -13682.315,E2 -13682.315} C_VEL
LIN {X 0,Y 348.051,Z 467.619,A -85,B 0,C 180,E1 -13686.96,E2 -13686.96} C_VEL
LIN {X 0,Y 347.885,Z 467.627,A -85,B 0,C 180,E1 -13690.477,E2 -13690.477} C_VEL
LIN {X 0,Y 347.85,Z 467.654,A -85,B 0,C 180,E1 -13694.12,E2 -13694.12} C_VEL
LIN {X 0,Y 347.786,Z 467.634,A -85,B 0,C 180,E1 -13698.239,E2 -13698.239} C_VEL
LIN {X 0,Y 347.762,Z 467.661,A -85,B 0,C 180,E1 -13701.625,E2 -13701.625} C_VEL
LIN {X 0,Y 347.737,Z 467.658,A -85,B 0,C 180,E1 -13705.116,E2 -13705.116} C_VEL
LIN {X 0,Y 347.728,Z 467.651,A -85,B 0,C 180,E1 -13707.703,E2 -13707.703} C_VEL
LIN {X 0,Y 347.739,Z 467.669,A -85,B 0,C 180,E1 -13710.35,E2 -13710.35} C_VEL
LIN {X 0,Y 347.749,Z 467.65,A -85,B 0,C 180,E1 -13714.045,E2 -13714.045} C_VEL
LIN {X 0,Y 347.755,Z 467.667,A -85,B 0,C 180,E1 -13717.323,E2 -13717.323} C_VEL
LIN {X 0,Y 347.697,Z 467.666,A -85,B 0,C 180,E1 -13720.304,E2 -13720.304} C_VEL
LIN {X 0,Y 347.722,Z 467.668,A -85,B 0,C 180,E1 -13723.41,E2 -13723.41} C_VEL
LIN {X 0,Y 347.724,Z 467.669,A -85,B 0,C 180,E1 -13726.688,E2 -13726.688} C_VEL
LIN {X 0,Y 347.703,Z 467.656,A -85,B 0,C 180,E1 -13730.184,E2 -13730.184} C_VEL
LIN {X 0,Y 347.757,Z 467.662,A -85,B 0,C 180,E1 -13732.679,E2 -13732.679} C_VEL
LIN {X 0,Y 347.752,Z 467.667,A -85,B 0,C 180,E1 -13735.957,E2 -13735.957} C_VEL
LIN {X 0,Y 347.795,Z 467.807,A -85,B 0,C 180,E1 -13737.62,E2 -13737.62} C_VEL
LIN {X 0,Y 349.445,Z 475.948,A -85,B 0,C 180,E1 -13740.57,E2 -13740.57} C_VEL
LIN {X 0,Y 351.066,Z 485.078,A -85,B 0,C 180,E1 -13743.55,E2 -13743.55} C_VEL
LIN {X 0,Y 350.626,Z 490.008,A -85,B 0,C 180,E1 -13745.107,E2 -13745.107} C_VEL
LIN {X 0,Y 349.996,Z 495.894,A -85,B 0,C 180,E1 -13746.915,E2 -13746.915} C_VEL
LIN {X 0,Y 350.866,Z 500.352,A -85,B 0,C 180,E1 -13747.134,E2 -13747.134} C_VEL
LIN {X 0,Y 355.258,Z 522.753,A -85,B 0,C 180,E1 -13747.909,E2 -13747.909} C_VEL
LIN {X 0,Y 356.893,Z 533.392,A -85,B 0,C 180,E1 -13748.24,E2 -13748.24} C_VEL
LIN {X 0,Y 355.706,Z 600.856,A -85,B 0,C 180,E1 -13749.621,E2 -13749.621} C_VEL
LIN {X 0,Y 355.21,Z 610.763,A -85,B 0,C 180,E1 -13749.931,E2 -13749.931} C_VEL
LIN {X 0,Y 354.64,Z 620.752,A -85,B 0,C 180,E1 -13750.388,E2 -13750.388} C_VEL
LIN {X 0,Y 353.744,Z 631.106,A -85,B 0,C 180,E1 -13751.015,E2 -13751.015} C_VEL
LIN {X 0,Y 352.929,Z 640.253,A -85,B 0,C 180,E1 -13751.722,E2 -13751.722} C_VEL
LIN {X 0,Y 351.959,Z 649.255,A -85,B 0,C 180,E1 -13752.571,E2 -13752.571} C_VEL
LIN {X 0,Y 350.988,Z 657.982,A -85,B 0,C 180,E1 -13753.571,E2 -13753.571} C_VEL
LIN {X 0,Y 350.121,Z 665.883,A -85,B 0,C 180,E1 -13754.652,E2 -13754.652} C_VEL
LIN {X 0,Y 349.111,Z 674.203,A -85,B 0,C 180,E1 -13756.021,E2 -13756.021} C_VEL
LIN {X 0,Y 348.38,Z 680.194,A -85,B 0,C 180,E1 -13757.179,E2 -13757.179} C_VEL
LIN {X 0,Y 347.565,Z 686.504,A -85,B 0,C 180,E1 -13758.63,E2 -13758.63} C_VEL
LIN {X 0,Y 347.035,Z 691.78,A -85,B 0,C 180,E1 -13760.088,E2 -13760.088} C_VEL
LIN {X 0,Y 346.572,Z 696.875,A -85,B 0,C 180,E1 -13761.839,E2 -13761.839} C_VEL
LIN {X 0,Y 346.246,Z 700.84,A -85,B 0,C 180,E1 -13763.591,E2 -13763.591} C_VEL
LIN {X 0,Y 346.161,Z 703.775,A -85,B 0,C 180,E1 -13765.342,E2 -13765.342} C_VEL
LIN {X 0,Y 346.144,Z 705.276,A -85,B 0,C 180,E1 -13766.508,E2 -13766.508} C_VEL
LIN {X 0,Y 346.105,Z 706.798,A -85,B 0,C 180,E1 -13768.836,E2 -13768.836} C_VEL
LIN {X 0,Y 346.15,Z 707.078,A -85,B 0,C 180,E1 -13770,E2 -13770} C_VEL
LIN {X 0,Y 346.086,Z 706.202,A -85,B 0,C 180,E1 -13772.328,E2 -13772.328} C_VEL
LIN {X 0,Y 346.144,Z 705.276,A -85,B 0,C 180,E1 -13773.492,E2 -13773.492} C_VEL
LIN {X 0,Y 346.202,Z 701.818,A -85,B 0,C 180,E1 -13775.885,E2 -13775.885} C_VEL
LIN {X 0,Y 346.472,Z 698.303,A -85,B 0,C 180,E1 -13777.576,E2 -13777.576} C_VEL
LIN {X 0,Y 346.87,Z 693.571,A -85,B 0,C 180,E1 -13779.328,E2 -13779.328} C_VEL
LIN {X 0,Y 347.469,Z 687.598,A -85,B 0,C 180,E1 -13781.078,E2 -13781.078} C_VEL
LIN {X 0,Y 348.005,Z 682.817,A -85,B 0,C 180,E1 -13782.242,E2 -13782.242} C_VEL
LIN {X 0,Y 348.744,Z 677.326,A -85,B 0,C 180,E1 -13783.4,E2 -13783.4} C_VEL
LIN {X 0,Y 349.752,Z 669.108,A -85,B 0,C 180,E1 -13784.845,E2 -13784.845} C_VEL
LIN {X 0,Y 350.678,Z 660.772,A -85,B 0,C 180,E1 -13786.064,E2 -13786.064} C_VEL
LIN {X 0,Y 351.537,Z 653.194,A -85,B 0,C 180,E1 -13787.001,E2 -13787.001} C_VEL
LIN {X 0,Y 352.574,Z 643.432,A -85,B 0,C 180,E1 -13787.997,E2 -13787.997} C_VEL
LIN {X 0,Y 353.45,Z 635.044,A -85,B 0,C 180,E1 -13788.701,E2 -13788.701} C_VEL
LIN {X 0,Y 354.343,Z 624.539,A -85,B 0,C 180,E1 -13789.403,E2 -13789.403} C_VEL
LIN {X 0,Y 354.951,Z 614.204,A -85,B 0,C 180,E1 -13789.933,E2 -13789.933} C_VEL
LIN {X 0,Y 355.587,Z 603.489,A -85,B 0,C 180,E1 -13790.311,E2 -13790.311} C_VEL
LIN {X 0,Y 356.147,Z 579.619,A -85,B 0,C 180,E1 -13790.829,E2 -13790.829} C_VEL
LIN {X 0,Y 356.809,Z 532.326,A -85,B 0,C 180,E1 -13791.788,E2 -13791.788} C_VEL
LIN {X 0,Y 352.524,Z 508.211,A -85,B 0,C 180,E1 -13792.584,E2 -13792.584} C_VEL
LIN {X 0,Y 349.959,Z 496.172,A -85,B 0,C 180,E1 -13793.05,E2 -13793.05} C_VEL
LIN {X 0,Y 350.024,Z 494.822,A -85,B 0,C 180,E1 -13793.363,E2 -13793.363} C_VEL
LIN {X 0,Y 351.115,Z 486.088,A -85,B 0,C 180,E1 -13796.126,E2 -13796.126} C_VEL
LIN {X 0,Y 350.12,Z 479.438,A -85,B 0,C 180,E1 -13798.339,E2 -13798.339} C_VEL
LIN {X 0,Y 348.225,Z 469.718,A -85,B 0,C 180,E1 -13801.65,E2 -13801.65} C_VEL
LIN {X 0,Y 347.785,Z 467.742,A -85,B 0,C 180,E1 -13802.454,E2 -13802.454} C_VEL
LIN {X 0,Y 347.769,Z 467.652,A -85,B 0,C 180,E1 -13806.063,E2 -13806.063} C_VEL
LIN {X 0,Y 347.733,Z 467.668,A -85,B 0,C 180,E1 -13808.795,E2 -13808.795} C_VEL
LIN {X 0,Y 347.742,Z 467.649,A -85,B 0,C 180,E1 -13811.831,E2 -13811.831} C_VEL
LIN {X 0,Y 347.7,Z 467.67,A -85,B 0,C 180,E1 -13815.027,E2 -13815.027} C_VEL
LIN {X 0,Y 347.74,Z 467.668,A -85,B 0,C 180,E1 -13818.399,E2 -13818.399} C_VEL
LIN {X 0,Y 347.762,Z 467.664,A -85,B 0,C 180,E1 -13822.013,E2 -13822.013} C_VEL
LIN {X 0,Y 347.744,Z 467.653,A -85,B 0,C 180,E1 -13825.534,E2 -13825.534} C_VEL
LIN {X 0,Y 347.746,Z 467.666,A -85,B 0,C 180,E1 -13828.299,E2 -13828.299} C_VEL
LIN {X 0,Y 347.745,Z 467.662,A -85,B 0,C 180,E1 -13830.983,E2 -13830.983} C_VEL
LIN {X 0,Y 347.734,Z 467.645,A -85,B 0,C 180,E1 -13833.598,E2 -13833.598} C_VEL
LIN {X 0,Y 347.748,Z 467.664,A -85,B 0,C 180,E1 -13836.157,E2 -13836.157} C_VEL
LIN {X 0,Y 347.737,Z 467.652,A -85,B 0,C 180,E1 -13839.903,E2 -13839.903} C_VEL
LIN {X 0,Y 347.795,Z 467.636,A -85,B 0,C 180,E1 -13842.354,E2 -13842.354} C_VEL
LIN {X 0,Y 347.85,Z 467.655,A -85,B 0,C 180,E1 -13845.967,E2 -13845.967} C_VEL
LIN {X 0,Y 347.885,Z 467.627,A -85,B 0,C 180,E1 -13849.523,E2 -13849.523} C_VEL
LIN {X 0,Y 348.051,Z 467.619,A -85,B 0,C 180,E1 -13853.04,E2 -13853.04} C_VEL
LIN {X 0,Y 348.176,Z 467.607,A -85,B 0,C 180,E1 -13857.685,E2 -13857.685} C_VEL
LIN {X 0,Y 348.111,Z 467.594,A -85,B 0,C 180,E1 -13861.155,E2 -13861.155} C_VEL
LIN {X 0,Y 348.175,Z 467.596,A -85,B 0,C 180,E1 -13862.312,E2 -13862.312} C_VEL
LIN {X 0,Y 348.046,Z 467.624,A -85,B 0,C 180,E1 -13866.957,E2 -13866.957} C_VEL
LIN {X 0,Y 347.883,Z 467.622,A -85,B 0,C 180,E1 -13870.474,E2 -13870.474} C_VEL
LIN {X 0,Y 347.873,Z 467.653,A -85,B 0,C 180,E1 -13874.135,E2 -13874.135} C_VEL
LIN {X 0,Y 347.78,Z 467.64,A -85,B 0,C 180,E1 -13878.236,E2 -13878.236} C_VEL
LIN {X 0,Y 347.758,Z 467.657,A -85,B 0,C 180,E1 -13881.624,E2 -13881.624} C_VEL
LIN {X 0,Y 347.73,Z 467.665,A -85,B 0,C 180,E1 -13885.112,E2 -13885.112} C_VEL
LIN {X 0,Y 347.714,Z 467.649,A -85,B 0,C 180,E1 -13887.7,E2 -13887.7} C_VEL
LIN {X 0,Y 347.728,Z 467.672,A -85,B 0,C 180,E1 -13890.347,E2 -13890.347} C_VEL
LIN {X 0,Y 347.737,Z 467.654,A -85,B 0,C 180,E1 -13894.042,E2 -13894.042} C_VEL
LIN {X 0,Y 347.743,Z 467.667,A -85,B 0,C 180,E1 -13897.32,E2 -13897.32} C_VEL
LIN {X 0,Y 347.683,Z 467.662,A -85,B 0,C 180,E1 -13900.301,E2 -13900.301} C_VEL
LIN {X 0,Y 347.708,Z 467.672,A -85,B 0,C 180,E1 -13903.407,E2 -13903.407} C_VEL
LIN {X 0,Y 347.709,Z 467.64,A -85,B 0,C 180,E1 -13906.686,E2 -13906.686} C_VEL
LIN {X 0,Y 347.687,Z 467.658,A -85,B 0,C 180,E1 -13910.181,E2 -13910.181} C_VEL
LIN {X 0,Y 347.74,Z 467.667,A -85,B 0,C 180,E1 -13912.677,E2 -13912.677} C_VEL
LIN {X 0,Y 347.734,Z 467.643,A -85,B 0,C 180,E1 -13915.955,E2 -13915.955} C_VEL
LIN {X 0,Y 347.724,Z 467.658,A -85,B 0,C 180,E1 -13919.65,E2 -13919.65} C_VEL
LIN {X 0,Y 347.721,Z 467.674,A -85,B 0,C 180,E1 -13923.599,E2 -13923.599} C_VEL
LIN {X 0,Y 347.737,Z 467.672,A -85,B 0,C 180,E1 -13926.158,E2 -13926.158} C_VEL
LIN {X 0,Y 347.796,Z 467.789,A -85,B 0,C 180,E1 -13929.136,E2 -13929.136} C_VEL
LIN {X 0,Y 348.014,Z 468.81,A -85,B 0,C 180,E1 -13929.459,E2 -13929.459} C_VEL
LIN {X 0,Y 349.58,Z 471.612,A -85,B 0,C 180,E1 -13929.904,E2 -13929.904} C_VEL
LIN {X 0,Y 351.788,Z 473.493,A -85,B 0,C 180,E1 -13930.406,E2 -13930.406} C_VEL
LIN {X 0,Y 353.903,Z 476.761,A -85,B 0,C 180,E1 -13930.989,E2 -13930.989} C_VEL
LIN {X 0,Y 356.522,Z 479.174,A -85,B 0,C 180,E1 -13931.642,E2 -13931.642} C_VEL
LIN {X 0,Y 358.921,Z 482.428,A -85,B 0,C 180,E1 -13932.322,E2 -13932.322} C_VEL
LIN {X 0,Y 361.691,Z 484.897,A -85,B 0,C 180,E1 -13933.078,E2 -13933.078} C_VEL
LIN {X 0,Y 364.37,Z 488.223,A -85,B 0,C 180,E1 -13933.898,E2 -13933.898} C_VEL
LIN {X 0,Y 367.926,Z 491.118,A -85,B 0,C 180,E1 -13934.968,E2 -13934.968} C_VEL
LIN {X 0,Y 371.006,Z 494.695,A -85,B 0,C 180,E1 -13936.037,E2 -13936.037} C_VEL
LIN {X 0,Y 374.477,Z 497.508,A -85,B 0,C 180,E1 -13937.295,E2 -13937.295} C_VEL
LIN {X 0,Y 377.29,Z 500.699,A -85,B 0,C 180,E1 -13938.456,E2 -13938.456} C_VEL
LIN {X 0,Y 380.196,Z 502.925,A -85,B 0,C 180,E1 -13939.729,E2 -13939.729} C_VEL
LIN {X 0,Y 382.271,Z 504.156,A -85,B 0,C 180,E1 -13940.715,E2 -13940.715} C_VEL
LIN {X 0,Y 385.028,Z 507.535,A -85,B 0,C 180,E1 -13942.374,E2 -13942.374} C_VEL
LIN {X 0,Y 387.576,Z 509.539,A -85,B 0,C 180,E1 -13944.25,E2 -13944.25} C_VEL
LIN {X 0,Y 389.258,Z 510.39,A -85,B 0,C 180,E1 -13945.859,E2 -13945.859} C_VEL
LIN {X 0,Y 390.387,Z 510.809,A -85,B 0,C 180,E1 -13947.437,E2 -13947.437} C_VEL
LIN {X 0,Y 390.949,Z 511.279,A -85,B 0,C 180,E1 -13948.97,E2 -13948.97} C_VEL
LIN {X 0,Y 391.111,Z 511.297,A -85,B 0,C 180,E1 -13950,E2 -13950} C_VEL
LIN {X 0,Y 390.766,Z 511.039,A -85,B 0,C 180,E1 -13951.787,E2 -13951.787} C_VEL
LIN {X 0,Y 389.564,Z 510.47,A -85,B 0,C 180,E1 -13953.765,E2 -13953.765} C_VEL
LIN {X 0,Y 388.142,Z 509.909,A -85,B 0,C 180,E1 -13955.234,E2 -13955.234} C_VEL
LIN {X 0,Y 386.068,Z 508.441,A -85,B 0,C 180,E1 -13956.887,E2 -13956.887} C_VEL
LIN {X 0,Y 384.077,Z 506.539,A -85,B 0,C 180,E1 -13958.194,E2 -13958.194} C_VEL
LIN {X 0,Y 381.742,Z 503.76,A -85,B 0,C 180,E1 -13959.537,E2 -13959.537} C_VEL
LIN {X 0,Y 378.657,Z 501.857,A -85,B 0,C 180,E1 -13960.967,E2 -13960.967} C_VEL
LIN {X 0,Y 375.452,Z 498.705,A -85,B 0,C 180,E1 -13962.328,E2 -13962.328} C_VEL
LIN {X 0,Y 373.825,Z 496.83,A -85,B 0,C 180,E1 -13962.954,E2 -13962.954} C_VEL
LIN {X 0,Y 370.717,Z 494.438,A -85,B 0,C 180,E1 -13964.059,E2 -13964.059} C_VEL
LIN {X 0,Y 367.766,Z 490.875,A -85,B 0,C 180,E1 -13965.087,E2 -13965.087} C_VEL
LIN {X 0,Y 363.79,Z 487.631,A -85,B 0,C 180,E1 -13966.282,E2 -13966.282} C_VEL
LIN {X 0,Y 361.067,Z 484.225,A -85,B 0,C 180,E1 -13967.094,E2 -13967.094} C_VEL
LIN {X 0,Y 358.127,Z 481.532,A -85,B 0,C 180,E1 -13967.907,E2 -13967.907} C_VEL
LIN {X 0,Y 355.796,Z 478.385,A -85,B 0,C 180,E1 -13968.541,E2 -13968.541} C_VEL
LIN {X 0,Y 353.181,Z 475.896,A -85,B 0,C 180,E1 -13969.202,E2 -13969.202} C_VEL
LIN {X 0,Y 351.272,Z 472.94,A -85,B 0,C 180,E1 -13969.719,E2 -13969.719} C_VEL
LIN {X 0,Y 349.005,Z 470.883,A -85,B 0,C 180,E1 -13970.234,E2 -13970.234} C_VEL
LIN {X 0,Y 347.889,Z 468.358,A -85,B 0,C 180,E1 -13970.626,E2 -13970.626} C_VEL
LIN {X 0,Y 347.785,Z 467.703,A -85,B 0,C 180,E1 -13971.02,E2 -13971.02} C_VEL
LIN {X 0,Y 347.724,Z 467.673,A -85,B 0,C 180,E1 -13975.115,E2 -13975.115} C_VEL
LIN {X 0,Y 347.71,Z 467.669,A -85,B 0,C 180,E1 -13977.702,E2 -13977.702} C_VEL
LIN {X 0,Y 347.724,Z 467.658,A -85,B 0,C 180,E1 -13980.35,E2 -13980.35} C_VEL
LIN {X 0,Y 347.734,Z 467.643,A -85,B 0,C 180,E1 -13984.045,E2 -13984.045} C_VEL
LIN {X 0,Y 347.74,Z 467.667,A -85,B 0,C 180,E1 -13987.323,E2 -13987.323} C_VEL
LIN {X 0,Y 347.682,Z 467.652,A -85,B 0,C 180,E1 -13990.304,E2 -13990.304} C_VEL
LIN {X 0,Y 347.707,Z 467.642,A -85,B 0,C 180,E1 -13993.41,E2 -13993.41} C_VEL
LIN {X 0,Y 347.71,Z 467.672,A -85,B 0,C 180,E1 -13996.688,E2 -13996.688} C_VEL
LIN {X 0,Y 347.689,Z 467.666,A -85,B 0,C 180,E1 -14000.184,E2 -14000.184} C_VEL
LIN {X 0,Y 347.743,Z 467.667,A -85,B 0,C 180,E1 -14002.68,E2 -14002.68} C_VEL
LIN {X 0,Y 347.737,Z 467.654,A -85,B 0,C 180,E1 -14005.958,E2 -14005.958} C_VEL
LIN {X 0,Y 347.72,Z 467.672,A -85,B 0,C 180,E1 -14009.526,E2 -14009.526} C_VEL
LIN {X 0,Y 347.087,Z 467.754,A -85,B 0,C 180,E1 -14010.494,E2 -14010.494} C_VEL
LIN {X 0,Y 344.216,Z 468.107,A -85,B 0,C 180,E1 -14012.067,E2 -14012.067} C_VEL
LIN {X 0,Y 341.772,Z 468.404,A -85,B 0,C 180,E1 -14013.34,E2 -14013.34} C_VEL
LIN {X 0,Y 340.74,Z 468.531,A -85,B 0,C 180,E1 -14014.327,E2 -14014.327} C_VEL
LIN {X 0,Y 340.668,Z 468.541,A -85,B 0,C 180,E1 -14014.661,E2 -14014.661} C_VEL
LIN {X 0,Y 340.715,Z 468.535,A -85,B 0,C 180,E1 -14018.207,E2 -14018.207} C_VEL
LIN {X 0,Y 340.744,Z 468.518,A -85,B 0,C 180,E1 -14021.98,E2 -14021.98} C_VEL
LIN {X 0,Y 340.826,Z 468.532,A -85,B 0,C 180,E1 -14025.732,E2 -14025.732} C_VEL
LIN {X 0,Y 340.836,Z 468.5,A -85,B 0,C 180,E1 -14029.307,E2 -14029.307} C_VEL
LIN {X 0,Y 340.994,Z 468.503,A -85,B 0,C 180,E1 -14032.898,E2 -14032.898} C_VEL
LIN {X 0,Y 340.801,Z 468.532,A -85,B 0,C 180,E1 -14035.27,E2 -14035.27} C_VEL
LIN {X 0,Y 341.112,Z 468.476,A -85,B 0,C 180,E1 -14037.64,E2 -14037.64} C_VEL
LIN {X 0,Y 341.082,Z 468.478,A -85,B 0,C 180,E1 -14041.182,E2 -14041.182} C_VEL
LIN {X 0,Y 341.113,Z 468.488,A -85,B 0,C 180,E1 -14042.363,E2 -14042.363} C_VEL
LIN {X 0,Y 341.008,Z 468.503,A -85,B 0,C 180,E1 -14045.916,E2 -14045.916} C_VEL
LIN {X 0,Y 340.961,Z 468.484,A -85,B 0,C 180,E1 -14048.358,E2 -14048.358} C_VEL
LIN {X 0,Y 340.831,Z 468.517,A -85,B 0,C 180,E1 -14051.902,E2 -14051.902} C_VEL
LIN {X 0,Y 340.809,Z 468.529,A -85,B 0,C 180,E1 -14054.329,E2 -14054.329} C_VEL
LIN {X 0,Y 340.749,Z 468.509,A -85,B 0,C 180,E1 -14058.423,E2 -14058.423} C_VEL
LIN {X 0,Y 340.718,Z 468.54,A -85,B 0,C 180,E1 -14061.843,E2 -14061.843} C_VEL
LIN {X 0,Y 340.67,Z 468.529,A -85,B 0,C 180,E1 -14065.674,E2 -14065.674} C_VEL
LIN {X 0,Y 340.679,Z 468.537,A -85,B 0,C 180,E1 -14068.327,E2 -14068.327} C_VEL
LIN {X 0,Y 340.694,Z 468.545,A -85,B 0,C 180,E1 -14071.047,E2 -14071.047} C_VEL
LIN {X 0,Y 340.716,Z 468.533,A -85,B 0,C 180,E1 -14075.281,E2 -14075.281} C_VEL
LIN {X 0,Y 340.694,Z 468.54,A -85,B 0,C 180,E1 -14078.383,E2 -14078.383} C_VEL
LIN {X 0,Y 340.692,Z 468.549,A -85,B 0,C 180,E1 -14082.045,E2 -14082.045} C_VEL
LIN {X 0,Y 340.651,Z 468.553,A -85,B 0,C 180,E1 -14086.229,E2 -14086.229} C_VEL
LIN {X 0,Y 340.67,Z 468.526,A -85,B 0,C 180,E1 -14088.689,E2 -14088.689} C_VEL
LIN {X 0,Y 340.721,Z 468.546,A -85,B 0,C 180,E1 -14091.772,E2 -14091.772} C_VEL
LIN {X 0,Y 340.726,Z 468.544,A -85,B 0,C 180,E1 -14095.597,E2 -14095.597} C_VEL
LIN {X 0,Y 340.754,Z 468.732,A -85,B 0,C 180,E1 -14097.265,E2 -14097.265} C_VEL
LIN {X 0,Y 342.311,Z 476.319,A -85,B 0,C 180,E1 -14100.078,E2 -14100.078} C_VEL
LIN {X 0,Y 343.883,Z 484.889,A -85,B 0,C 180,E1 -14102.953,E2 -14102.953} C_VEL
LIN {X 0,Y 344.103,Z 487.949,A -85,B 0,C 180,E1 -14103.985,E2 -14103.985} C_VEL
LIN {X 0,Y 343.15,Z 495.614,A -85,B 0,C 180,E1 -14106.411,E2 -14106.411} C_VEL
LIN {X 0,Y 343.54,Z 497.945,A -85,B 0,C 180,E1 -14106.569,E2 -14106.569} C_VEL
LIN {X 0,Y 347.875,Z 519.399,A -85,B 0,C 180,E1 -14107.346,E2 -14107.346} C_VEL
LIN {X 0,Y 350.315,Z 534.245,A -85,B 0,C 180,E1 -14107.832,E2 -14107.832} C_VEL
LIN {X 0,Y 349.071,Z 600.667,A -85,B 0,C 180,E1 -14109.216,E2 -14109.216} C_VEL
LIN {X 0,Y 348.56,Z 610.567,A -85,B 0,C 180,E1 -14109.531,E2 -14109.531} C_VEL
LIN {X 0,Y 347.943,Z 620.555,A -85,B 0,C 180,E1 -14109.994,E2 -14109.994} C_VEL
LIN {X 0,Y 347.046,Z 630.91,A -85,B 0,C 180,E1 -14110.634,E2 -14110.634} C_VEL
LIN {X 0,Y 346.199,Z 640.057,A -85,B 0,C 180,E1 -14111.354,E2 -14111.354} C_VEL
LIN {X 0,Y 345.165,Z 649.057,A -85,B 0,C 180,E1 -14112.217,E2 -14112.217} C_VEL
LIN {X 0,Y 344.148,Z 657.785,A -85,B 0,C 180,E1 -14113.235,E2 -14113.235} C_VEL
LIN {X 0,Y 343.177,Z 666.357,A -85,B 0,C 180,E1 -14114.444,E2 -14114.444} C_VEL
LIN {X 0,Y 342.185,Z 674.006,A -85,B 0,C 180,E1 -14115.732,E2 -14115.732} C_VEL
LIN {X 0,Y 341.43,Z 679.997,A -85,B 0,C 180,E1 -14116.914,E2 -14116.914} C_VEL
LIN {X 0,Y 340.57,Z 686.307,A -85,B 0,C 180,E1 -14118.393,E2 -14118.393} C_VEL
LIN {X 0,Y 340.03,Z 691.583,A -85,B 0,C 180,E1 -14119.882,E2 -14119.882} C_VEL
LIN {X 0,Y 339.532,Z 696.678,A -85,B 0,C 180,E1 -14121.669,E2 -14121.669} C_VEL
LIN {X 0,Y 339.171,Z 700.642,A -85,B 0,C 180,E1 -14123.456,E2 -14123.456} C_VEL
LIN {X 0,Y 339.064,Z 703.578,A -85,B 0,C 180,E1 -14125.244,E2 -14125.244} C_VEL
LIN {X 0,Y 339.068,Z 705.08,A -85,B 0,C 180,E1 -14126.435,E2 -14126.435} C_VEL
LIN {X 0,Y 339.008,Z 706.602,A -85,B 0,C 180,E1 -14128.812,E2 -14128.812} C_VEL
LIN {X 0,Y 339.052,Z 706.882,A -85,B 0,C 180,E1 -14130,E2 -14130} C_VEL
LIN {X 0,Y 339,Z 706.006,A -85,B 0,C 180,E1 -14132.376,E2 -14132.376} C_VEL
LIN {X 0,Y 339.068,Z 705.08,A -85,B 0,C 180,E1 -14133.565,E2 -14133.565} C_VEL
LIN {X 0,Y 339.118,Z 701.731,A -85,B 0,C 180,E1 -14135.948,E2 -14135.948} C_VEL
LIN {X 0,Y 339.405,Z 698.106,A -85,B 0,C 180,E1 -14137.735,E2 -14137.735} C_VEL
LIN {X 0,Y 339.824,Z 693.373,A -85,B 0,C 180,E1 -14139.523,E2 -14139.523} C_VEL
LIN {X 0,Y 340.464,Z 687.4,A -85,B 0,C 180,E1 -14141.309,E2 -14141.309} C_VEL
LIN {X 0,Y 341.056,Z 682.62,A -85,B 0,C 180,E1 -14142.496,E2 -14142.496} C_VEL
LIN {X 0,Y 341.822,Z 677.129,A -85,B 0,C 180,E1 -14143.677,E2 -14143.677} C_VEL
LIN {X 0,Y 342.888,Z 668.912,A -85,B 0,C 180,E1 -14145.149,E2 -14145.149} C_VEL
LIN {X 0,Y 343.795,Z 660.783,A -85,B 0,C 180,E1 -14146.366,E2 -14146.366} C_VEL
LIN {X 0,Y 344.739,Z 652.997,A -85,B 0,C 180,E1 -14147.346,E2 -14147.346} C_VEL
LIN {X 0,Y 345.817,Z 643.236,A -85,B 0,C 180,E1 -14148.361,E2 -14148.361} C_VEL
LIN {X 0,Y 346.725,Z 634.848,A -85,B 0,C 180,E1 -14149.077,E2 -14149.077} C_VEL
LIN {X 0,Y 347.662,Z 624.343,A -85,B 0,C 180,E1 -14149.791,E2 -14149.791} C_VEL
LIN {X 0,Y 348.295,Z 614.008,A -85,B 0,C 180,E1 -14150.331,E2 -14150.331} C_VEL
LIN {X 0,Y 348.953,Z 603.293,A -85,B 0,C 180,E1 -14150.714,E2 -14150.714} C_VEL
LIN {X 0,Y 349.521,Z 579.504,A -85,B 0,C 180,E1 -14151.241,E2 -14151.241} C_VEL
LIN {X 0,Y 350.3,Z 533.789,A -85,B 0,C 180,E1 -14152.178,E2 -14152.178} C_VEL
LIN {X 0,Y 346.143,Z 510.216,A -85,B 0,C 180,E1 -14152.975,E2 -14152.975} C_VEL
LIN {X 0,Y 343.109,Z 495.902,A -85,B 0,C 180,E1 -14153.545,E2 -14153.545} C_VEL
LIN {X 0,Y 343.33,Z 493.677,A -85,B 0,C 180,E1 -14154.167,E2 -14154.167} C_VEL
LIN {X 0,Y 344.149,Z 487.166,A -85,B 0,C 180,E1 -14156.271,E2 -14156.271} C_VEL
LIN {X 0,Y 342.985,Z 479.755,A -85,B 0,C 180,E1 -14158.81,E2 -14158.81} C_VEL
LIN {X 0,Y 341.41,Z 471.744,A -85,B 0,C 180,E1 -14161.62,E2 -14161.62} C_VEL
LIN {X 0,Y 340.757,Z 468.643,A -85,B 0,C 180,E1 -14162.778,E2 -14162.778} C_VEL
LIN {X 0,Y 340.703,Z 468.534,A -85,B 0,C 180,E1 -14166.741,E2 -14166.741} C_VEL
LIN {X 0,Y 340.652,Z 468.529,A -85,B 0,C 180,E1 -14170.238,E2 -14170.238} C_VEL
LIN {X 0,Y 340.674,Z 468.547,A -85,B 0,C 180,E1 -14172.904,E2 -14172.904} C_VEL
LIN {X 0,Y 340.674,Z 468.547,A -85,B 0,C 180,E1 -14177.094,E2 -14177.094} C_VEL
LIN {X 0,Y 340.656,Z 468.54,A -85,B 0,C 180,E1 -14180.24,E2 -14180.24} C_VEL
LIN {X 0,Y 340.708,Z 468.545,A -85,B 0,C 180,E1 -14183.559,E2 -14183.559} C_VEL
LIN {X 0,Y 340.693,Z 468.529,A -85,B 0,C 180,E1 -14186.152,E2 -14186.152} C_VEL
LIN {X 0,Y 340.722,Z 468.544,A -85,B 0,C 180,E1 -14190.033,E2 -14190.033} C_VEL
LIN {X 0,Y 340.71,Z 468.52,A -85,B 0,C 180,E1 -14193.01,E2 -14193.01} C_VEL
LIN {X 0,Y 340.699,Z 468.542,A -85,B 0,C 180,E1 -14196.923,E2 -14196.923} C_VEL
LIN {X 0,Y 340.688,Z 468.521,A -85,B 0,C 180,E1 -14200.726,E2 -14200.726} C_VEL
LIN {X 0,Y 340.718,Z 468.526,A -85,B 0,C 180,E1 -14203.213,E2 -14203.213} C_VEL
LIN {X 0,Y 340.812,Z 468.526,A -85,B 0,C 180,E1 -14206.888,E2 -14206.888} C_VEL
LIN {X 0,Y 340.877,Z 468.49,A -85,B 0,C 180,E1 -14210.505,E2 -14210.505} C_VEL
LIN {X 0,Y 340.998,Z 468.498,A -85,B 0,C 180,E1 -14212.895,E2 -14212.895} C_VEL
LIN {X 0,Y 340.802,Z 468.531,A -85,B 0,C 180,E1 -14215.267,E2 -14215.267} C_VEL
LIN {X 0,Y 341.113,Z 468.488,A -85,B 0,C 180,E1 -14217.637,E2 -14217.637} C_VEL
LIN {X 0,Y 341.082,Z 468.469,A -85,B 0,C 180,E1 -14221.179,E2 -14221.179} C_VEL
LIN {X 0,Y 341.112,Z 468.476,A -85,B 0,C 180,E1 -14222.36,E2 -14222.36} C_VEL
LIN {X 0,Y 340.981,Z 468.506,A -85,B 0,C 180,E1 -14226.531,E2 -14226.531} C_VEL
LIN {X 0,Y 340.874,Z 468.496,A -85,B 0,C 180,E1 -14229.492,E2 -14229.492} C_VEL
LIN {X 0,Y 340.833,Z 468.522,A -85,B 0,C 180,E1 -14233.108,E2 -14233.108} C_VEL
LIN {X 0,Y 340.722,Z 468.534,A -85,B 0,C 180,E1 -14236.783,E2 -14236.783} C_VEL
LIN {X 0,Y 340.682,Z 468.518,A -85,B 0,C 180,E1 -14239.271,E2 -14239.271} C_VEL
LIN {X 0,Y 340.696,Z 468.544,A -85,B 0,C 180,E1 -14243.073,E2 -14243.073} C_VEL
LIN {X 0,Y 340.7,Z 468.523,A -85,B 0,C 180,E1 -14246.986,E2 -14246.986} C_VEL
LIN {X 0,Y 340.683,Z 468.547,A -85,B 0,C 180,E1 -14251.044,E2 -14251.044} C_VEL
LIN {X 0,Y 340.704,Z 468.53,A -85,B 0,C 180,E1 -14255.278,E2 -14255.278} C_VEL
LIN {X 0,Y 340.681,Z 468.548,A -85,B 0,C 180,E1 -14258.381,E2 -14258.381} C_VEL
LIN {X 0,Y 340.678,Z 468.541,A -85,B 0,C 180,E1 -14262.042,E2 -14262.042} C_VEL
LIN {X 0,Y 340.636,Z 468.527,A -85,B 0,C 180,E1 -14266.226,E2 -14266.226} C_VEL
LIN {X 0,Y 340.636,Z 468.529,A -85,B 0,C 180,E1 -14269.76,E2 -14269.76} C_VEL
LIN {X 0,Y 340.686,Z 468.542,A -85,B 0,C 180,E1 -14273.257,E2 -14273.257} C_VEL
LIN {X 0,Y 340.678,Z 468.523,A -85,B 0,C 180,E1 -14276.152,E2 -14276.152} C_VEL
LIN {X 0,Y 340.707,Z 468.527,A -85,B 0,C 180,E1 -14280.034,E2 -14280.034} C_VEL
LIN {X 0,Y 340.696,Z 468.548,A -85,B 0,C 180,E1 -14283.011,E2 -14283.011} C_VEL
LIN {X 0,Y 340.691,Z 468.549,A -85,B 0,C 180,E1 -14286.925,E2 -14286.925} C_VEL
LIN {X 0,Y 340.746,Z 468.784,A -85,B 0,C 180,E1 -14287.897,E2 -14287.897} C_VEL
LIN {X 0,Y 341.018,Z 469.911,A -85,B 0,C 180,E1 -14288.162,E2 -14288.162} C_VEL
LIN {X 0,Y 342.631,Z 472.571,A -85,B 0,C 180,E1 -14288.57,E2 -14288.57} C_VEL
LIN {X 0,Y 344.479,Z 474.31,A -85,B 0,C 180,E1 -14288.959,E2 -14288.959} C_VEL
LIN {X 0,Y 346.705,Z 477.658,A -85,B 0,C 180,E1 -14289.516,E2 -14289.516} C_VEL
LIN {X 0,Y 348.878,Z 479.783,A -85,B 0,C 180,E1 -14290.022,E2 -14290.022} C_VEL
LIN {X 0,Y 351.575,Z 483.259,A -85,B 0,C 180,E1 -14290.686,E2 -14290.686} C_VEL
LIN {X 0,Y 353.742,Z 485.342,A -85,B 0,C 180,E1 -14291.24,E2 -14291.24} C_VEL
